  [680] = {x=33.236, y=0.000, z=-5.463, rx=-0.000, ry=0.000, rz=-0.000, shoulder=lefty, elbow=epositive, wrist=wnegative, fatherId=fReference[0]}
  [681] = {x=32.701, y=0.000, z=-5.454, rx=-0.000, ry=0.000, rz=-0.000, shoulder=lefty, elbow=epositive, wrist=wnegative, fatherId=fReference[0]}
  [682] = {x=32.182, y=0.000, z=-5.451, rx=-0.000, ry=0.000, rz=-0.000, shoulder=lefty, elbow=epositive, wrist=wnegative, fatherId=fReference[0]}
  [683] = {x=31.672, y=0.000, z=-5.452, rx=-0.000, ry=0.000, rz=-0.000, shoulder=lefty, elbow=epositive, wrist=wnegative, fatherId=fReference[0]}
  [684] = {x=31.165, y=0.000, z=-5.456, rx=-0.000, ry=0.000, rz=-0.000, shoulder=lefty, elbow=epositive, wrist=wnegative, fatherId=fReference[0]}
  [685] = {x=30.661, y=0.000, z=-5.462, rx=-0.000, ry=0.000, rz=-0.000, shoulder=lefty, elbow=epositive, wrist=wnegative, fatherId=fReference[0]}
  [686] = {x=30.158, y=0.000, z=-5.467, rx=-0.000, ry=0.000, rz=-0.000, shoulder=lefty, elbow=epositive, wrist=wnegative, fatherId=fReference[0]}
  [687] = {x=29.655, y=0.000, z=-5.473, rx=-0.000, ry=0.000, rz=-0.000, shoulder=lefty, elbow=epositive, wrist=wnegative, fatherId=fReference[0]}
  [688] = {x=29.154, y=0.000, z=-5.480, rx=-0.000, ry=0.000, rz=-0.000, shoulder=lefty, elbow=epositive, wrist=wnegative, fatherId=fReference[0]}
  [689] = {x=28.652, y=0.000, z=-5.487, rx=-0.000, ry=0.000, rz=-0.000, shoulder=lefty, elbow=epositive, wrist=wnegative, fatherId=fReference[0]}
  [690] = {x=28.151, y=0.000, z=-5.494, rx=-0.000, ry=0.000, rz=-0.000, shoulder=lefty, elbow=epositive, wrist=wnegative, fatherId=fReference[0]}
  [691] = {x=27.650, y=0.000, z=-5.502, rx=-0.000, ry=0.000, rz=-0.000, shoulder=lefty, elbow=epositive, wrist=wnegative, fatherId=fReference[0]}
  [692] = {x=27.149, y=0.000, z=-5.510, rx=-0.000, ry=0.000, rz=-0.000, shoulder=lefty, elbow=epositive, wrist=wnegative, fatherId=fReference[0]}
  [693] = {x=26.649, y=0.000, z=-5.518, rx=-0.000, ry=0.000, rz=-0.000, shoulder=lefty, elbow=epositive, wrist=wnegative, fatherId=fReference[0]}
  [694] = {x=26.149, y=0.000, z=-5.526, rx=-0.000, ry=0.000, rz=-0.000, shoulder=lefty, elbow=epositive, wrist=wnegative, fatherId=fReference[0]}
  [695] = {x=25.648, y=0.000, z=-5.534, rx=-0.000, ry=0.000, rz=-0.000, shoulder=lefty, elbow=epositive, wrist=wnegative, fatherId=fReference[0]}
  [696] = {x=25.148, y=0.000, z=-5.543, rx=-0.000, ry=0.000, rz=-0.000, shoulder=lefty, elbow=epositive, wrist=wnegative, fatherId=fReference[0]}
  [697] = {x=24.648, y=0.000, z=-5.551, rx=-0.000, ry=0.000, rz=-0.000, shoulder=lefty, elbow=epositive, wrist=wnegative, fatherId=fReference[0]}
  [698] = {x=24.148, y=0.000, z=-5.559, rx=-0.000, ry=0.000, rz=-0.000, shoulder=lefty, elbow=epositive, wrist=wnegative, fatherId=fReference[0]}
  [699] = {x=23.647, y=0.000, z=-5.568, rx=-0.000, ry=0.000, rz=-0.000, shoulder=lefty, elbow=epositive, wrist=wnegative, fatherId=fReference[0]}
  [700] = {x=23.147, y=0.000, z=-5.576, rx=-0.000, ry=0.000, rz=-0.000, shoulder=lefty, elbow=epositive, wrist=wnegative, fatherId=fReference[0]}
  [701] = {x=22.647, y=0.000, z=-5.585, rx=-0.000, ry=0.000, rz=-0.000, shoulder=lefty, elbow=epositive, wrist=wnegative, fatherId=fReference[0]}
  [702] = {x=22.147, y=0.000, z=-5.594, rx=-0.000, ry=0.000, rz=-0.000, shoulder=lefty, elbow=epositive, wrist=wnegative, fatherId=fReference[0]}
  [703] = {x=21.647, y=0.000, z=-5.602, rx=-0.000, ry=0.000, rz=-0.000, shoulder=lefty, elbow=epositive, wrist=wnegative, fatherId=fReference[0]}
  [704] = {x=21.146, y=0.000, z=-5.611, rx=-0.000, ry=0.000, rz=-0.000, shoulder=lefty, elbow=epositive, wrist=wnegative, fatherId=fReference[0]}
  [705] = {x=20.646, y=0.000, z=-5.620, rx=-0.000, ry=0.000, rz=-0.000, shoulder=lefty, elbow=epositive, wrist=wnegative, fatherId=fReference[0]}
  [706] = {x=20.146, y=0.000, z=-5.629, rx=-0.000, ry=0.000, rz=-0.000, shoulder=lefty, elbow=epositive, wrist=wnegative, fatherId=fReference[0]}
  [707] = {x=19.646, y=0.000, z=-5.638, rx=-0.000, ry=0.000, rz=-0.000, shoulder=lefty, elbow=epositive, wrist=wnegative, fatherId=fReference[0]}
  [708] = {x=19.146, y=0.000, z=-5.647, rx=-0.000, ry=0.000, rz=-0.000, shoulder=lefty, elbow=epositive, wrist=wnegative, fatherId=fReference[0]}
  [709] = {x=18.646, y=0.000, z=-5.656, rx=-0.000, ry=0.000, rz=-0.000, shoulder=lefty, elbow=epositive, wrist=wnegative, fatherId=fReference[0]}
  [710] = {x=18.145, y=0.000, z=-5.665, rx=-0.000, ry=0.000, rz=-0.000, shoulder=lefty, elbow=epositive, wrist=wnegative, fatherId=fReference[0]}
  [711] = {x=17.645, y=0.000, z=-5.675, rx=-0.000, ry=0.000, rz=-0.000, shoulder=lefty, elbow=epositive, wrist=wnegative, fatherId=fReference[0]}
  [712] = {x=17.145, y=0.000, z=-5.684, rx=-0.000, ry=0.000, rz=-0.000, shoulder=lefty, elbow=epositive, wrist=wnegative, fatherId=fReference[0]}
  [713] = {x=16.645, y=0.000, z=-5.693, rx=-0.000, ry=0.000, rz=-0.000, shoulder=lefty, elbow=epositive, wrist=wnegative, fatherId=fReference[0]}
  [714] = {x=16.144, y=0.000, z=-5.702, rx=-0.000, ry=0.000, rz=-0.000, shoulder=lefty, elbow=epositive, wrist=wnegative, fatherId=fReference[0]}
  [715] = {x=15.644, y=0.000, z=-5.712, rx=-0.000, ry=0.000, rz=-0.000, shoulder=lefty, elbow=epositive, wrist=wnegative, fatherId=fReference[0]}
  [716] = {x=15.144, y=0.000, z=-5.721, rx=-0.000, ry=0.000, rz=-0.000, shoulder=lefty, elbow=epositive, wrist=wnegative, fatherId=fReference[0]}
  [717] = {x=14.644, y=0.000, z=-5.730, rx=-0.000, ry=0.000, rz=-0.000, shoulder=lefty, elbow=epositive, wrist=wnegative, fatherId=fReference[0]}
  [718] = {x=14.144, y=0.000, z=-5.740, rx=-0.000, ry=0.000, rz=-0.000, shoulder=lefty, elbow=epositive, wrist=wnegative, fatherId=fReference[0]}
  [719] = {x=13.643, y=0.000, z=-5.749, rx=-0.000, ry=0.000, rz=-0.000, shoulder=lefty, elbow=epositive, wrist=wnegative, fatherId=fReference[0]}
  [720] = {x=13.143, y=0.000, z=-5.758, rx=-0.000, ry=0.000, rz=-0.000, shoulder=lefty, elbow=epositive, wrist=wnegative, fatherId=fReference[0]}
  [721] = {x=12.643, y=0.000, z=-5.767, rx=-0.000, ry=0.000, rz=-0.000, shoulder=lefty, elbow=epositive, wrist=wnegative, fatherId=fReference[0]}
  [722] = {x=12.142, y=0.000, z=-5.776, rx=-0.000, ry=0.000, rz=-0.000, shoulder=lefty, elbow=epositive, wrist=wnegative, fatherId=fReference[0]}
  [723] = {x=11.641, y=0.000, z=-5.785, rx=-0.000, ry=0.000, rz=-0.000, shoulder=lefty, elbow=epositive, wrist=wnegative, fatherId=fReference[0]}
  [724] = {x=11.141, y=0.000, z=-5.794, rx=-0.000, ry=0.000, rz=-0.000, shoulder=lefty, elbow=epositive, wrist=wnegative, fatherId=fReference[0]}
  [725] = {x=10.640, y=0.000, z=-5.803, rx=-0.000, ry=0.000, rz=-0.000, shoulder=lefty, elbow=epositive, wrist=wnegative, fatherId=fReference[0]}
  [726] = {x=10.139, y=0.000, z=-5.811, rx=-0.000, ry=0.000, rz=-0.000, shoulder=lefty, elbow=epositive, wrist=wnegative, fatherId=fReference[0]}
  [727] = {x=9.638, y=0.000, z=-5.820, rx=-0.000, ry=0.000, rz=-0.000, shoulder=lefty, elbow=epositive, wrist=wnegative, fatherId=fReference[0]}
  [728] = {x=9.137, y=0.000, z=-5.828, rx=-0.000, ry=0.000, rz=-0.000, shoulder=lefty, elbow=epositive, wrist=wnegative, fatherId=fReference[0]}
  [729] = {x=8.637, y=0.000, z=-5.837, rx=-0.000, ry=0.000, rz=-0.000, shoulder=lefty, elbow=epositive, wrist=wnegative, fatherId=fReference[0]}
  [730] = {x=8.136, y=0.000, z=-5.846, rx=-0.000, ry=0.000, rz=-0.000, shoulder=lefty, elbow=epositive, wrist=wnegative, fatherId=fReference[0]}
  [731] = {x=7.635, y=0.000, z=-5.854, rx=-0.000, ry=0.000, rz=-0.000, shoulder=lefty, elbow=epositive, wrist=wnegative, fatherId=fReference[0]}
  [732] = {x=7.134, y=0.000, z=-5.862, rx=-0.000, ry=0.000, rz=-0.000, shoulder=lefty, elbow=epositive, wrist=wnegative, fatherId=fReference[0]}
  [733] = {x=6.633, y=0.000, z=-5.870, rx=-0.000, ry=0.000, rz=-0.000, shoulder=lefty, elbow=epositive, wrist=wnegative, fatherId=fReference[0]}
  [734] = {x=6.131, y=0.000, z=-5.878, rx=-0.000, ry=0.000, rz=-0.000, shoulder=lefty, elbow=epositive, wrist=wnegative, fatherId=fReference[0]}
  [735] = {x=5.630, y=0.000, z=-5.886, rx=-0.000, ry=0.000, rz=-0.000, shoulder=lefty, elbow=epositive, wrist=wnegative, fatherId=fReference[0]}
  [736] = {x=5.128, y=0.000, z=-5.894, rx=-0.000, ry=0.000, rz=-0.000, shoulder=lefty, elbow=epositive, wrist=wnegative, fatherId=fReference[0]}
  [737] = {x=4.626, y=0.000, z=-5.902, rx=-0.000, ry=0.000, rz=-0.000, shoulder=lefty, elbow=epositive, wrist=wnegative, fatherId=fReference[0]}
  [738] = {x=4.123, y=0.000, z=-5.909, rx=-0.000, ry=0.000, rz=-0.000, shoulder=lefty, elbow=epositive, wrist=wnegative, fatherId=fReference[0]}
  [739] = {x=3.621, y=0.000, z=-5.917, rx=-0.000, ry=0.000, rz=-0.000, shoulder=lefty, elbow=epositive, wrist=wnegative, fatherId=fReference[0]}
  [740] = {x=3.120, y=0.000, z=-5.925, rx=-0.000, ry=0.000, rz=-0.000, shoulder=lefty, elbow=epositive, wrist=wnegative, fatherId=fReference[0]}
  [741] = {x=2.618, y=0.000, z=-5.932, rx=-0.000, ry=0.000, rz=-0.000, shoulder=lefty, elbow=epositive, wrist=wnegative, fatherId=fReference[0]}
  [742] = {x=2.117, y=0.000, z=-5.941, rx=-0.000, ry=0.000, rz=-0.000, shoulder=lefty, elbow=epositive, wrist=wnegative, fatherId=fReference[0]}
  [743] = {x=1.616, y=0.000, z=-5.949, rx=-0.000, ry=0.000, rz=-0.000, shoulder=lefty, elbow=epositive, wrist=wnegative, fatherId=fReference[0]}
  [744] = {x=1.114, y=0.000, z=-5.957, rx=-0.000, ry=0.000, rz=-0.000, shoulder=lefty, elbow=epositive, wrist=wnegative, fatherId=fReference[0]}
  [745] = {x=0.614, y=0.000, z=-5.966, rx=-0.000, ry=0.000, rz=-0.000, shoulder=lefty, elbow=epositive, wrist=wnegative, fatherId=fReference[0]}
  [746] = {x=0.112, y=0.000, z=-5.974, rx=-0.000, ry=0.000, rz=-0.000, shoulder=lefty, elbow=epositive, wrist=wnegative, fatherId=fReference[0]}
  [747] = {x=-0.389, y=0.000, z=-5.983, rx=-0.000, ry=0.000, rz=-0.000, shoulder=lefty, elbow=epositive, wrist=wnegative, fatherId=fReference[0]}
  [748] = {x=-0.890, y=0.000, z=-5.991, rx=-0.000, ry=0.000, rz=-0.000, shoulder=lefty, elbow=epositive, wrist=wnegative, fatherId=fReference[0]}
  [749] = {x=-1.392, y=0.000, z=-6.000, rx=-0.000, ry=0.000, rz=-0.000, shoulder=lefty, elbow=epositive, wrist=wnegative, fatherId=fReference[0]}
  [750] = {x=-1.893, y=0.000, z=-6.009, rx=-0.000, ry=0.000, rz=-0.000, shoulder=lefty, elbow=epositive, wrist=wnegative, fatherId=fReference[0]}
  [751] = {x=-2.394, y=0.000, z=-6.017, rx=-0.000, ry=0.000, rz=-0.000, shoulder=lefty, elbow=epositive, wrist=wnegative, fatherId=fReference[0]}
  [752] = {x=-2.895, y=0.000, z=-6.026, rx=-0.000, ry=0.000, rz=-0.000, shoulder=lefty, elbow=epositive, wrist=wnegative, fatherId=fReference[0]}
  [753] = {x=-3.397, y=0.000, z=-6.035, rx=-0.000, ry=0.000, rz=-0.000, shoulder=lefty, elbow=epositive, wrist=wnegative, fatherId=fReference[0]}
  [754] = {x=-3.898, y=0.000, z=-6.044, rx=-0.000, ry=0.000, rz=-0.000, shoulder=lefty, elbow=epositive, wrist=wnegative, fatherId=fReference[0]}
  [755] = {x=-4.399, y=0.000, z=-6.053, rx=-0.000, ry=0.000, rz=-0.000, shoulder=lefty, elbow=epositive, wrist=wnegative, fatherId=fReference[0]}
  [756] = {x=-4.901, y=0.000, z=-6.062, rx=-0.000, ry=0.000, rz=-0.000, shoulder=lefty, elbow=epositive, wrist=wnegative, fatherId=fReference[0]}
  [757] = {x=-5.402, y=0.000, z=-6.071, rx=-0.000, ry=0.000, rz=-0.000, shoulder=lefty, elbow=epositive, wrist=wnegative, fatherId=fReference[0]}
  [758] = {x=-5.902, y=0.000, z=-6.080, rx=-0.000, ry=0.000, rz=-0.000, shoulder=lefty, elbow=epositive, wrist=wnegative, fatherId=fReference[0]}
  [759] = {x=-6.404, y=0.000, z=-6.089, rx=-0.000, ry=0.000, rz=-0.000, shoulder=lefty, elbow=epositive, wrist=wnegative, fatherId=fReference[0]}
  [760] = {x=-6.906, y=0.000, z=-6.098, rx=-0.000, ry=0.000, rz=-0.000, shoulder=lefty, elbow=epositive, wrist=wnegative, fatherId=fReference[0]}
  [761] = {x=-7.407, y=0.000, z=-6.107, rx=-0.000, ry=0.000, rz=-0.000, shoulder=lefty, elbow=epositive, wrist=wnegative, fatherId=fReference[0]}
  [762] = {x=-7.907, y=0.000, z=-6.117, rx=-0.000, ry=0.000, rz=-0.000, shoulder=lefty, elbow=epositive, wrist=wnegative, fatherId=fReference[0]}
  [763] = {x=-8.409, y=0.000, z=-6.126, rx=-0.000, ry=0.000, rz=-0.000, shoulder=lefty, elbow=epositive, wrist=wnegative, fatherId=fReference[0]}
  [764] = {x=-8.910, y=0.000, z=-6.136, rx=-0.000, ry=0.000, rz=-0.000, shoulder=lefty, elbow=epositive, wrist=wnegative, fatherId=fReference[0]}
  [765] = {x=-9.411, y=0.000, z=-6.145, rx=-0.000, ry=0.000, rz=-0.000, shoulder=lefty, elbow=epositive, wrist=wnegative, fatherId=fReference[0]}
  [766] = {x=-9.912, y=0.000, z=-6.155, rx=-0.000, ry=0.000, rz=-0.000, shoulder=lefty, elbow=epositive, wrist=wnegative, fatherId=fReference[0]}
  [767] = {x=-10.412, y=0.000, z=-6.165, rx=-0.000, ry=0.000, rz=-0.000, shoulder=lefty, elbow=epositive, wrist=wnegative, fatherId=fReference[0]}
  [768] = {x=-10.913, y=0.000, z=-6.175, rx=-0.000, ry=0.000, rz=-0.000, shoulder=lefty, elbow=epositive, wrist=wnegative, fatherId=fReference[0]}
  [769] = {x=-11.413, y=0.000, z=-6.185, rx=-0.000, ry=0.000, rz=-0.000, shoulder=lefty, elbow=epositive, wrist=wnegative, fatherId=fReference[0]}
  [770] = {x=-11.914, y=0.000, z=-6.195, rx=-0.000, ry=0.000, rz=-0.000, shoulder=lefty, elbow=epositive, wrist=wnegative, fatherId=fReference[0]}
  [771] = {x=-12.414, y=0.000, z=-6.206, rx=-0.000, ry=0.000, rz=-0.000, shoulder=lefty, elbow=epositive, wrist=wnegative, fatherId=fReference[0]}
  [772] = {x=-12.916, y=0.000, z=-6.215, rx=-0.000, ry=0.000, rz=-0.000, shoulder=lefty, elbow=epositive, wrist=wnegative, fatherId=fReference[0]}
  [773] = {x=-13.416, y=0.000, z=-6.225, rx=-0.000, ry=0.000, rz=-0.000, shoulder=lefty, elbow=epositive, wrist=wnegative, fatherId=fReference[0]}
  [774] = {x=-13.916, y=0.000, z=-6.236, rx=-0.000, ry=0.000, rz=-0.000, shoulder=lefty, elbow=epositive, wrist=wnegative, fatherId=fReference[0]}
  [775] = {x=-14.417, y=0.000, z=-6.246, rx=-0.000, ry=0.000, rz=-0.000, shoulder=lefty, elbow=epositive, wrist=wnegative, fatherId=fReference[0]}
  [776] = {x=-14.916, y=0.000, z=-6.257, rx=-0.000, ry=0.000, rz=-0.000, shoulder=lefty, elbow=epositive, wrist=wnegative, fatherId=fReference[0]}
  [777] = {x=-15.418, y=0.000, z=-6.267, rx=-0.000, ry=0.000, rz=-0.000, shoulder=lefty, elbow=epositive, wrist=wnegative, fatherId=fReference[0]}
  [778] = {x=-15.917, y=0.000, z=-6.278, rx=-0.000, ry=0.000, rz=-0.000, shoulder=lefty, elbow=epositive, wrist=wnegative, fatherId=fReference[0]}
  [779] = {x=-16.418, y=0.000, z=-6.288, rx=-0.000, ry=0.000, rz=-0.000, shoulder=lefty, elbow=epositive, wrist=wnegative, fatherId=fReference[0]}
  [780] = {x=-16.918, y=0.000, z=-6.300, rx=-0.000, ry=0.000, rz=-0.000, shoulder=lefty, elbow=epositive, wrist=wnegative, fatherId=fReference[0]}
  [781] = {x=-17.419, y=0.000, z=-6.310, rx=-0.000, ry=0.000, rz=-0.000, shoulder=lefty, elbow=epositive, wrist=wnegative, fatherId=fReference[0]}
  [782] = {x=-17.919, y=0.000, z=-6.321, rx=-0.000, ry=0.000, rz=-0.000, shoulder=lefty, elbow=epositive, wrist=wnegative, fatherId=fReference[0]}
  [783] = {x=-18.420, y=0.000, z=-6.331, rx=-0.000, ry=0.000, rz=-0.000, shoulder=lefty, elbow=epositive, wrist=wnegative, fatherId=fReference[0]}
  [784] = {x=-18.920, y=0.000, z=-6.342, rx=-0.000, ry=0.000, rz=-0.000, shoulder=lefty, elbow=epositive, wrist=wnegative, fatherId=fReference[0]}
  [785] = {x=-19.418, y=0.000, z=-6.354, rx=-0.000, ry=0.000, rz=-0.000, shoulder=lefty, elbow=epositive, wrist=wnegative, fatherId=fReference[0]}
  [786] = {x=-19.920, y=0.000, z=-6.364, rx=-0.000, ry=0.000, rz=-0.000, shoulder=lefty, elbow=epositive, wrist=wnegative, fatherId=fReference[0]}
  [787] = {x=-20.420, y=0.000, z=-6.375, rx=-0.000, ry=0.000, rz=-0.000, shoulder=lefty, elbow=epositive, wrist=wnegative, fatherId=fReference[0]}
  [788] = {x=-20.920, y=0.000, z=-6.386, rx=-0.000, ry=0.000, rz=-0.000, shoulder=lefty, elbow=epositive, wrist=wnegative, fatherId=fReference[0]}
  [789] = {x=-21.421, y=0.000, z=-6.397, rx=-0.000, ry=0.000, rz=-0.000, shoulder=lefty, elbow=epositive, wrist=wnegative, fatherId=fReference[0]}
  [790] = {x=-21.922, y=0.000, z=-6.407, rx=-0.000, ry=0.000, rz=-0.000, shoulder=lefty, elbow=epositive, wrist=wnegative, fatherId=fReference[0]}
  [791] = {x=-22.422, y=0.000, z=-6.418, rx=-0.000, ry=0.000, rz=-0.000, shoulder=lefty, elbow=epositive, wrist=wnegative, fatherId=fReference[0]}
  [792] = {x=-22.921, y=0.000, z=-6.431, rx=-0.000, ry=0.000, rz=-0.000, shoulder=lefty, elbow=epositive, wrist=wnegative, fatherId=fReference[0]}
  [793] = {x=-23.422, y=0.000, z=-6.442, rx=-0.000, ry=0.000, rz=-0.000, shoulder=lefty, elbow=epositive, wrist=wnegative, fatherId=fReference[0]}
  [794] = {x=-23.924, y=0.000, z=-6.453, rx=-0.000, ry=0.000, rz=-0.000, shoulder=lefty, elbow=epositive, wrist=wnegative, fatherId=fReference[0]}
  [795] = {x=-24.426, y=0.000, z=-6.464, rx=-0.000, ry=0.000, rz=-0.000, shoulder=lefty, elbow=epositive, wrist=wnegative, fatherId=fReference[0]}
  [796] = {x=-24.927, y=0.000, z=-6.476, rx=-0.000, ry=0.000, rz=-0.000, shoulder=lefty, elbow=epositive, wrist=wnegative, fatherId=fReference[0]}
  [797] = {x=-25.427, y=0.000, z=-6.488, rx=-0.000, ry=0.000, rz=-0.000, shoulder=lefty, elbow=epositive, wrist=wnegative, fatherId=fReference[0]}
  [798] = {x=-25.928, y=0.000, z=-6.501, rx=-0.000, ry=0.000, rz=-0.000, shoulder=lefty, elbow=epositive, wrist=wnegative, fatherId=fReference[0]}
  [799] = {x=-26.428, y=0.000, z=-6.513, rx=-0.000, ry=0.000, rz=-0.000, shoulder=lefty, elbow=epositive, wrist=wnegative, fatherId=fReference[0]}
  [800] = {x=-26.930, y=0.000, z=-6.526, rx=-0.000, ry=0.000, rz=-0.000, shoulder=lefty, elbow=epositive, wrist=wnegative, fatherId=fReference[0]}
  [801] = {x=-27.433, y=0.000, z=-6.538, rx=-0.000, ry=0.000, rz=-0.000, shoulder=lefty, elbow=epositive, wrist=wnegative, fatherId=fReference[0]}
  [802] = {x=-27.936, y=0.000, z=-6.550, rx=-0.000, ry=0.000, rz=-0.000, shoulder=lefty, elbow=epositive, wrist=wnegative, fatherId=fReference[0]}
  [803] = {x=-28.441, y=0.000, z=-6.561, rx=-0.000, ry=0.000, rz=-0.000, shoulder=lefty, elbow=epositive, wrist=wnegative, fatherId=fReference[0]}
  [804] = {x=-28.947, y=0.000, z=-6.571, rx=-0.000, ry=0.000, rz=-0.000, shoulder=lefty, elbow=epositive, wrist=wnegative, fatherId=fReference[0]}
  [805] = {x=-29.456, y=0.000, z=-6.581, rx=-0.000, ry=0.000, rz=-0.000, shoulder=lefty, elbow=epositive, wrist=wnegative, fatherId=fReference[0]}
  [806] = {x=-29.968, y=0.000, z=-6.590, rx=-0.000, ry=0.000, rz=-0.000, shoulder=lefty, elbow=epositive, wrist=wnegative, fatherId=fReference[0]}
  [807] = {x=-30.478, y=0.000, z=-6.600, rx=-0.000, ry=0.000, rz=-0.000, shoulder=lefty, elbow=epositive, wrist=wnegative, fatherId=fReference[0]}
  [808] = {x=-30.992, y=0.000, z=-6.610, rx=-0.000, ry=0.000, rz=-0.000, shoulder=lefty, elbow=epositive, wrist=wnegative, fatherId=fReference[0]}
  [809] = {x=-31.504, y=0.000, z=-6.617, rx=-0.000, ry=0.000, rz=-0.000, shoulder=lefty, elbow=epositive, wrist=wnegative, fatherId=fReference[0]}
  [810] = {x=-31.724, y=0.000, z=-6.575, rx=-0.000, ry=0.000, rz=-0.000, shoulder=lefty, elbow=epositive, wrist=wnegative, fatherId=fReference[0]}
  [811] = {x=-31.202, y=0.000, z=-6.559, rx=-0.000, ry=0.000, rz=-0.000, shoulder=lefty, elbow=epositive, wrist=wnegative, fatherId=fReference[0]}
  [812] = {x=-30.687, y=0.000, z=-6.554, rx=-0.000, ry=0.000, rz=-0.000, shoulder=lefty, elbow=epositive, wrist=wnegative, fatherId=fReference[0]}
  [813] = {x=-30.181, y=0.000, z=-6.554, rx=-0.000, ry=0.000, rz=-0.000, shoulder=lefty, elbow=epositive, wrist=wnegative, fatherId=fReference[0]}
  [814] = {x=-29.680, y=0.000, z=-6.557, rx=-0.000, ry=0.000, rz=-0.000, shoulder=lefty, elbow=epositive, wrist=wnegative, fatherId=fReference[0]}
  [815] = {x=-29.180, y=0.000, z=-6.561, rx=-0.000, ry=0.000, rz=-0.000, shoulder=lefty, elbow=epositive, wrist=wnegative, fatherId=fReference[0]}
  [816] = {x=-28.680, y=0.000, z=-6.566, rx=-0.000, ry=0.000, rz=-0.000, shoulder=lefty, elbow=epositive, wrist=wnegative, fatherId=fReference[0]}
  [817] = {x=-28.180, y=0.000, z=-6.571, rx=-0.000, ry=0.000, rz=-0.000, shoulder=lefty, elbow=epositive, wrist=wnegative, fatherId=fReference[0]}
  [818] = {x=-27.680, y=0.000, z=-6.577, rx=-0.000, ry=0.000, rz=-0.000, shoulder=lefty, elbow=epositive, wrist=wnegative, fatherId=fReference[0]}
  [819] = {x=-27.180, y=0.000, z=-6.584, rx=-0.000, ry=0.000, rz=-0.000, shoulder=lefty, elbow=epositive, wrist=wnegative, fatherId=fReference[0]}
  [820] = {x=-26.679, y=0.000, z=-6.591, rx=-0.000, ry=0.000, rz=-0.000, shoulder=lefty, elbow=epositive, wrist=wnegative, fatherId=fReference[0]}
  [821] = {x=-26.178, y=0.000, z=-6.598, rx=-0.000, ry=0.000, rz=-0.000, shoulder=lefty, elbow=epositive, wrist=wnegative, fatherId=fReference[0]}
  [822] = {x=-25.677, y=0.000, z=-6.605, rx=-0.000, ry=0.000, rz=-0.000, shoulder=lefty, elbow=epositive, wrist=wnegative, fatherId=fReference[0]}
  [823] = {x=-25.175, y=0.000, z=-6.613, rx=-0.000, ry=0.000, rz=-0.000, shoulder=lefty, elbow=epositive, wrist=wnegative, fatherId=fReference[0]}
  [824] = {x=-24.675, y=0.000, z=-6.622, rx=-0.000, ry=0.000, rz=-0.000, shoulder=lefty, elbow=epositive, wrist=wnegative, fatherId=fReference[0]}
  [825] = {x=-24.174, y=0.000, z=-6.630, rx=-0.000, ry=0.000, rz=-0.000, shoulder=lefty, elbow=epositive, wrist=wnegative, fatherId=fReference[0]}
  [826] = {x=-23.672, y=0.000, z=-6.639, rx=-0.000, ry=0.000, rz=-0.000, shoulder=lefty, elbow=epositive, wrist=wnegative, fatherId=fReference[0]}
  [827] = {x=-23.171, y=0.000, z=-6.647, rx=-0.000, ry=0.000, rz=-0.000, shoulder=lefty, elbow=epositive, wrist=wnegative, fatherId=fReference[0]}
  [828] = {x=-22.670, y=0.000, z=-6.656, rx=-0.000, ry=0.000, rz=-0.000, shoulder=lefty, elbow=epositive, wrist=wnegative, fatherId=fReference[0]}
  [829] = {x=-22.168, y=0.000, z=-6.665, rx=-0.000, ry=0.000, rz=-0.000, shoulder=lefty, elbow=epositive, wrist=wnegative, fatherId=fReference[0]}
  [830] = {x=-21.666, y=0.000, z=-6.673, rx=-0.000, ry=0.000, rz=-0.000, shoulder=lefty, elbow=epositive, wrist=wnegative, fatherId=fReference[0]}
  [831] = {x=-21.165, y=0.000, z=-6.682, rx=-0.000, ry=0.000, rz=-0.000, shoulder=lefty, elbow=epositive, wrist=wnegative, fatherId=fReference[0]}
  [832] = {x=-20.664, y=0.000, z=-6.691, rx=-0.000, ry=0.000, rz=-0.000, shoulder=lefty, elbow=epositive, wrist=wnegative, fatherId=fReference[0]}
  [833] = {x=-20.162, y=0.000, z=-6.699, rx=-0.000, ry=0.000, rz=-0.000, shoulder=lefty, elbow=epositive, wrist=wnegative, fatherId=fReference[0]}
  [834] = {x=-19.661, y=0.000, z=-6.708, rx=-0.000, ry=0.000, rz=-0.000, shoulder=lefty, elbow=epositive, wrist=wnegative, fatherId=fReference[0]}
  [835] = {x=-19.159, y=0.000, z=-6.716, rx=-0.000, ry=0.000, rz=-0.000, shoulder=lefty, elbow=epositive, wrist=wnegative, fatherId=fReference[0]}
  [836] = {x=-18.657, y=0.000, z=-6.724, rx=-0.000, ry=0.000, rz=-0.000, shoulder=lefty, elbow=epositive, wrist=wnegative, fatherId=fReference[0]}
  [837] = {x=-18.156, y=0.000, z=-6.733, rx=-0.000, ry=0.000, rz=-0.000, shoulder=lefty, elbow=epositive, wrist=wnegative, fatherId=fReference[0]}
  [838] = {x=-17.654, y=0.000, z=-6.742, rx=-0.000, ry=0.000, rz=-0.000, shoulder=lefty, elbow=epositive, wrist=wnegative, fatherId=fReference[0]}
  [839] = {x=-17.152, y=0.000, z=-6.750, rx=-0.000, ry=0.000, rz=-0.000, shoulder=lefty, elbow=epositive, wrist=wnegative, fatherId=fReference[0]}
  [840] = {x=-16.651, y=0.000, z=-6.758, rx=-0.000, ry=0.000, rz=-0.000, shoulder=lefty, elbow=epositive, wrist=wnegative, fatherId=fReference[0]}
  [841] = {x=-16.149, y=0.000, z=-6.767, rx=-0.000, ry=0.000, rz=-0.000, shoulder=lefty, elbow=epositive, wrist=wnegative, fatherId=fReference[0]}
  [842] = {x=-15.647, y=0.000, z=-6.776, rx=-0.000, ry=0.000, rz=-0.000, shoulder=lefty, elbow=epositive, wrist=wnegative, fatherId=fReference[0]}
  [843] = {x=-15.146, y=0.000, z=-6.785, rx=-0.000, ry=0.000, rz=-0.000, shoulder=lefty, elbow=epositive, wrist=wnegative, fatherId=fReference[0]}
  [844] = {x=-14.643, y=0.000, z=-6.793, rx=-0.000, ry=0.000, rz=-0.000, shoulder=lefty, elbow=epositive, wrist=wnegative, fatherId=fReference[0]}
  [845] = {x=-14.141, y=0.000, z=-6.802, rx=-0.000, ry=0.000, rz=-0.000, shoulder=lefty, elbow=epositive, wrist=wnegative, fatherId=fReference[0]}
  [846] = {x=-13.639, y=0.000, z=-6.811, rx=-0.000, ry=0.000, rz=-0.000, shoulder=lefty, elbow=epositive, wrist=wnegative, fatherId=fReference[0]}
  [847] = {x=-13.138, y=0.000, z=-6.819, rx=-0.000, ry=0.000, rz=-0.000, shoulder=lefty, elbow=epositive, wrist=wnegative, fatherId=fReference[0]}
  [848] = {x=-12.636, y=0.000, z=-6.828, rx=-0.000, ry=0.000, rz=-0.000, shoulder=lefty, elbow=epositive, wrist=wnegative, fatherId=fReference[0]}
  [849] = {x=-12.134, y=0.000, z=-6.837, rx=-0.000, ry=0.000, rz=-0.000, shoulder=lefty, elbow=epositive, wrist=wnegative, fatherId=fReference[0]}
  [850] = {x=-11.632, y=0.000, z=-6.846, rx=-0.000, ry=0.000, rz=-0.000, shoulder=lefty, elbow=epositive, wrist=wnegative, fatherId=fReference[0]}
  [851] = {x=-11.130, y=0.000, z=-6.856, rx=-0.000, ry=0.000, rz=-0.000, shoulder=lefty, elbow=epositive, wrist=wnegative, fatherId=fReference[0]}
  [852] = {x=-10.627, y=0.000, z=-6.865, rx=-0.000, ry=0.000, rz=-0.000, shoulder=lefty, elbow=epositive, wrist=wnegative, fatherId=fReference[0]}
  [853] = {x=-10.124, y=0.000, z=-6.874, rx=-0.000, ry=0.000, rz=-0.000, shoulder=lefty, elbow=epositive, wrist=wnegative, fatherId=fReference[0]}
  [854] = {x=-9.622, y=0.000, z=-6.884, rx=-0.000, ry=0.000, rz=-0.000, shoulder=lefty, elbow=epositive, wrist=wnegative, fatherId=fReference[0]}
  [855] = {x=-9.120, y=0.000, z=-6.893, rx=-0.000, ry=0.000, rz=-0.000, shoulder=lefty, elbow=epositive, wrist=wnegative, fatherId=fReference[0]}
  [856] = {x=-8.617, y=0.000, z=-6.902, rx=-0.000, ry=0.000, rz=-0.000, shoulder=lefty, elbow=epositive, wrist=wnegative, fatherId=fReference[0]}
  [857] = {x=-8.114, y=0.000, z=-6.910, rx=-0.000, ry=0.000, rz=-0.000, shoulder=lefty, elbow=epositive, wrist=wnegative, fatherId=fReference[0]}
  [858] = {x=-7.611, y=0.000, z=-6.920, rx=-0.000, ry=0.000, rz=-0.000, shoulder=lefty, elbow=epositive, wrist=wnegative, fatherId=fReference[0]}
  [859] = {x=-7.109, y=0.000, z=-6.928, rx=-0.000, ry=0.000, rz=-0.000, shoulder=lefty, elbow=epositive, wrist=wnegative, fatherId=fReference[0]}
  [860] = {x=-6.606, y=0.000, z=-6.937, rx=-0.000, ry=0.000, rz=-0.000, shoulder=lefty, elbow=epositive, wrist=wnegative, fatherId=fReference[0]}
  [861] = {x=-6.104, y=0.000, z=-6.945, rx=-0.000, ry=0.000, rz=-0.000, shoulder=lefty, elbow=epositive, wrist=wnegative, fatherId=fReference[0]}
  [862] = {x=-5.601, y=0.000, z=-6.952, rx=-0.000, ry=0.000, rz=-0.000, shoulder=lefty, elbow=epositive, wrist=wnegative, fatherId=fReference[0]}
  [863] = {x=-5.099, y=0.000, z=-6.961, rx=-0.000, ry=0.000, rz=-0.000, shoulder=lefty, elbow=epositive, wrist=wnegative, fatherId=fReference[0]}
  [864] = {x=-4.597, y=0.000, z=-6.969, rx=-0.000, ry=0.000, rz=-0.000, shoulder=lefty, elbow=epositive, wrist=wnegative, fatherId=fReference[0]}
  [865] = {x=-4.094, y=0.000, z=-6.976, rx=-0.000, ry=0.000, rz=-0.000, shoulder=lefty, elbow=epositive, wrist=wnegative, fatherId=fReference[0]}
  [866] = {x=-3.592, y=0.000, z=-6.985, rx=-0.000, ry=0.000, rz=-0.000, shoulder=lefty, elbow=epositive, wrist=wnegative, fatherId=fReference[0]}
  [867] = {x=-3.090, y=0.000, z=-6.993, rx=-0.000, ry=0.000, rz=-0.000, shoulder=lefty, elbow=epositive, wrist=wnegative, fatherId=fReference[0]}
  [868] = {x=-2.587, y=0.000, z=-7.001, rx=-0.000, ry=0.000, rz=-0.000, shoulder=lefty, elbow=epositive, wrist=wnegative, fatherId=fReference[0]}
  [869] = {x=-2.084, y=0.000, z=-7.009, rx=-0.000, ry=0.000, rz=-0.000, shoulder=lefty, elbow=epositive, wrist=wnegative, fatherId=fReference[0]}
  [870] = {x=-1.581, y=0.000, z=-7.016, rx=-0.000, ry=0.000, rz=-0.000, shoulder=lefty, elbow=epositive, wrist=wnegative, fatherId=fReference[0]}
  [871] = {x=-1.078, y=0.000, z=-7.025, rx=-0.000, ry=0.000, rz=-0.000, shoulder=lefty, elbow=epositive, wrist=wnegative, fatherId=fReference[0]}
  [872] = {x=-0.576, y=0.000, z=-7.034, rx=-0.000, ry=0.000, rz=-0.000, shoulder=lefty, elbow=epositive, wrist=wnegative, fatherId=fReference[0]}
  [873] = {x=-0.073, y=0.000, z=-7.042, rx=-0.000, ry=0.000, rz=-0.000, shoulder=lefty, elbow=epositive, wrist=wnegative, fatherId=fReference[0]}
  [874] = {x=0.430, y=0.000, z=-7.050, rx=-0.000, ry=0.000, rz=-0.000, shoulder=lefty, elbow=epositive, wrist=wnegative, fatherId=fReference[0]}
  [875] = {x=0.933, y=0.000, z=-7.058, rx=-0.000, ry=0.000, rz=-0.000, shoulder=lefty, elbow=epositive, wrist=wnegative, fatherId=fReference[0]}
  [876] = {x=1.436, y=0.000, z=-7.067, rx=-0.000, ry=0.000, rz=-0.000, shoulder=lefty, elbow=epositive, wrist=wnegative, fatherId=fReference[0]}
  [877] = {x=1.939, y=0.000, z=-7.076, rx=-0.000, ry=0.000, rz=-0.000, shoulder=lefty, elbow=epositive, wrist=wnegative, fatherId=fReference[0]}
  [878] = {x=2.442, y=0.000, z=-7.085, rx=-0.000, ry=0.000, rz=-0.000, shoulder=lefty, elbow=epositive, wrist=wnegative, fatherId=fReference[0]}
  [879] = {x=2.945, y=0.000, z=-7.093, rx=-0.000, ry=0.000, rz=-0.000, shoulder=lefty, elbow=epositive, wrist=wnegative, fatherId=fReference[0]}
  [880] = {x=3.448, y=0.000, z=-7.102, rx=-0.000, ry=0.000, rz=-0.000, shoulder=lefty, elbow=epositive, wrist=wnegative, fatherId=fReference[0]}
  [881] = {x=3.951, y=0.000, z=-7.112, rx=-0.000, ry=0.000, rz=-0.000, shoulder=lefty, elbow=epositive, wrist=wnegative, fatherId=fReference[0]}
  [882] = {x=4.454, y=0.000, z=-7.121, rx=-0.000, ry=0.000, rz=-0.000, shoulder=lefty, elbow=epositive, wrist=wnegative, fatherId=fReference[0]}
  [883] = {x=4.957, y=0.000, z=-7.129, rx=-0.000, ry=0.000, rz=-0.000, shoulder=lefty, elbow=epositive, wrist=wnegative, fatherId=fReference[0]}
  [884] = {x=5.460, y=0.000, z=-7.138, rx=-0.000, ry=0.000, rz=-0.000, shoulder=lefty, elbow=epositive, wrist=wnegative, fatherId=fReference[0]}
  [885] = {x=5.963, y=0.000, z=-7.147, rx=-0.000, ry=0.000, rz=-0.000, shoulder=lefty, elbow=epositive, wrist=wnegative, fatherId=fReference[0]}
  [886] = {x=6.466, y=0.000, z=-7.157, rx=-0.000, ry=0.000, rz=-0.000, shoulder=lefty, elbow=epositive, wrist=wnegative, fatherId=fReference[0]}
  [887] = {x=6.968, y=0.000, z=-7.167, rx=-0.000, ry=0.000, rz=-0.000, shoulder=lefty, elbow=epositive, wrist=wnegative, fatherId=fReference[0]}
  [888] = {x=7.471, y=0.000, z=-7.176, rx=-0.000, ry=0.000, rz=-0.000, shoulder=lefty, elbow=epositive, wrist=wnegative, fatherId=fReference[0]}
  [889] = {x=7.975, y=0.000, z=-7.186, rx=-0.000, ry=0.000, rz=-0.000, shoulder=lefty, elbow=epositive, wrist=wnegative, fatherId=fReference[0]}
  [890] = {x=8.478, y=0.000, z=-7.196, rx=-0.000, ry=0.000, rz=-0.000, shoulder=lefty, elbow=epositive, wrist=wnegative, fatherId=fReference[0]}
  [891] = {x=8.981, y=0.000, z=-7.205, rx=-0.000, ry=0.000, rz=-0.000, shoulder=lefty, elbow=epositive, wrist=wnegative, fatherId=fReference[0]}
  [892] = {x=9.484, y=0.000, z=-7.215, rx=-0.000, ry=0.000, rz=-0.000, shoulder=lefty, elbow=epositive, wrist=wnegative, fatherId=fReference[0]}
  [893] = {x=9.986, y=0.000, z=-7.225, rx=-0.000, ry=0.000, rz=-0.000, shoulder=lefty, elbow=epositive, wrist=wnegative, fatherId=fReference[0]}
  [894] = {x=10.489, y=0.000, z=-7.236, rx=-0.000, ry=0.000, rz=-0.000, shoulder=lefty, elbow=epositive, wrist=wnegative, fatherId=fReference[0]}
  [895] = {x=10.991, y=0.000, z=-7.246, rx=-0.000, ry=0.000, rz=-0.000, shoulder=lefty, elbow=epositive, wrist=wnegative, fatherId=fReference[0]}
  [896] = {x=11.494, y=0.000, z=-7.256, rx=-0.000, ry=0.000, rz=-0.000, shoulder=lefty, elbow=epositive, wrist=wnegative, fatherId=fReference[0]}
  [897] = {x=11.998, y=0.000, z=-7.267, rx=-0.000, ry=0.000, rz=-0.000, shoulder=lefty, elbow=epositive, wrist=wnegative, fatherId=fReference[0]}
  [898] = {x=12.500, y=0.000, z=-7.277, rx=-0.000, ry=0.000, rz=-0.000, shoulder=lefty, elbow=epositive, wrist=wnegative, fatherId=fReference[0]}
  [899] = {x=13.003, y=0.000, z=-7.287, rx=-0.000, ry=0.000, rz=-0.000, shoulder=lefty, elbow=epositive, wrist=wnegative, fatherId=fReference[0]}
  [900] = {x=13.506, y=0.000, z=-7.298, rx=-0.000, ry=0.000, rz=-0.000, shoulder=lefty, elbow=epositive, wrist=wnegative, fatherId=fReference[0]}
  [901] = {x=14.010, y=0.000, z=-7.308, rx=-0.000, ry=0.000, rz=-0.000, shoulder=lefty, elbow=epositive, wrist=wnegative, fatherId=fReference[0]}
  [902] = {x=14.513, y=0.000, z=-7.319, rx=-0.000, ry=0.000, rz=-0.000, shoulder=lefty, elbow=epositive, wrist=wnegative, fatherId=fReference[0]}
  [903] = {x=15.017, y=0.000, z=-7.330, rx=-0.000, ry=0.000, rz=-0.000, shoulder=lefty, elbow=epositive, wrist=wnegative, fatherId=fReference[0]}
  [904] = {x=15.519, y=0.000, z=-7.341, rx=-0.000, ry=0.000, rz=-0.000, shoulder=lefty, elbow=epositive, wrist=wnegative, fatherId=fReference[0]}
  [905] = {x=16.024, y=0.000, z=-7.350, rx=-0.000, ry=0.000, rz=-0.000, shoulder=lefty, elbow=epositive, wrist=wnegative, fatherId=fReference[0]}
  [906] = {x=16.527, y=0.000, z=-7.361, rx=-0.000, ry=0.000, rz=-0.000, shoulder=lefty, elbow=epositive, wrist=wnegative, fatherId=fReference[0]}
  [907] = {x=17.030, y=0.000, z=-7.373, rx=-0.000, ry=0.000, rz=-0.000, shoulder=lefty, elbow=epositive, wrist=wnegative, fatherId=fReference[0]}
  [908] = {x=17.534, y=0.000, z=-7.383, rx=-0.000, ry=0.000, rz=-0.000, shoulder=lefty, elbow=epositive, wrist=wnegative, fatherId=fReference[0]}
  [909] = {x=18.037, y=0.000, z=-7.394, rx=-0.000, ry=0.000, rz=-0.000, shoulder=lefty, elbow=epositive, wrist=wnegative, fatherId=fReference[0]}
  [910] = {x=18.542, y=0.000, z=-7.405, rx=-0.000, ry=0.000, rz=-0.000, shoulder=lefty, elbow=epositive, wrist=wnegative, fatherId=fReference[0]}
  [911] = {x=19.046, y=0.000, z=-7.415, rx=-0.000, ry=0.000, rz=-0.000, shoulder=lefty, elbow=epositive, wrist=wnegative, fatherId=fReference[0]}
  [912] = {x=19.550, y=0.000, z=-7.428, rx=-0.000, ry=0.000, rz=-0.000, shoulder=lefty, elbow=epositive, wrist=wnegative, fatherId=fReference[0]}
  [913] = {x=20.055, y=0.000, z=-7.437, rx=-0.000, ry=0.000, rz=-0.000, shoulder=lefty, elbow=epositive, wrist=wnegative, fatherId=fReference[0]}
  [914] = {x=20.559, y=0.000, z=-7.450, rx=-0.000, ry=0.000, rz=-0.000, shoulder=lefty, elbow=epositive, wrist=wnegative, fatherId=fReference[0]}
  [915] = {x=21.062, y=0.000, z=-7.462, rx=-0.000, ry=0.000, rz=-0.000, shoulder=lefty, elbow=epositive, wrist=wnegative, fatherId=fReference[0]}
  [916] = {x=21.567, y=0.000, z=-7.473, rx=-0.000, ry=0.000, rz=-0.000, shoulder=lefty, elbow=epositive, wrist=wnegative, fatherId=fReference[0]}
  [917] = {x=22.072, y=0.000, z=-7.484, rx=-0.000, ry=0.000, rz=-0.000, shoulder=lefty, elbow=epositive, wrist=wnegative, fatherId=fReference[0]}
  [918] = {x=22.578, y=0.000, z=-7.493, rx=-0.000, ry=0.000, rz=-0.000, shoulder=lefty, elbow=epositive, wrist=wnegative, fatherId=fReference[0]}
  [919] = {x=23.082, y=0.000, z=-7.505, rx=-0.000, ry=0.000, rz=-0.000, shoulder=lefty, elbow=epositive, wrist=wnegative, fatherId=fReference[0]}
  [920] = {x=23.588, y=0.000, z=-7.515, rx=-0.000, ry=0.000, rz=-0.000, shoulder=lefty, elbow=epositive, wrist=wnegative, fatherId=fReference[0]}
  [921] = {x=24.093, y=0.000, z=-7.528, rx=-0.000, ry=0.000, rz=-0.000, shoulder=lefty, elbow=epositive, wrist=wnegative, fatherId=fReference[0]}
  [922] = {x=24.598, y=0.000, z=-7.540, rx=-0.000, ry=0.000, rz=-0.000, shoulder=lefty, elbow=epositive, wrist=wnegative, fatherId=fReference[0]}
  [923] = {x=25.104, y=0.000, z=-7.552, rx=-0.000, ry=0.000, rz=-0.000, shoulder=lefty, elbow=epositive, wrist=wnegative, fatherId=fReference[0]}
  [924] = {x=25.610, y=0.000, z=-7.563, rx=-0.000, ry=0.000, rz=-0.000, shoulder=lefty, elbow=epositive, wrist=wnegative, fatherId=fReference[0]}
  [925] = {x=26.118, y=0.000, z=-7.572, rx=-0.000, ry=0.000, rz=-0.000, shoulder=lefty, elbow=epositive, wrist=wnegative, fatherId=fReference[0]}
  [926] = {x=26.625, y=0.000, z=-7.583, rx=-0.000, ry=0.000, rz=-0.000, shoulder=lefty, elbow=epositive, wrist=wnegative, fatherId=fReference[0]}
  [927] = {x=27.133, y=0.000, z=-7.595, rx=-0.000, ry=0.000, rz=-0.000, shoulder=lefty, elbow=epositive, wrist=wnegative, fatherId=fReference[0]}
  [928] = {x=27.642, y=0.000, z=-7.608, rx=-0.000, ry=0.000, rz=-0.000, shoulder=lefty, elbow=epositive, wrist=wnegative, fatherId=fReference[0]}
  [929] = {x=28.150, y=0.000, z=-7.621, rx=-0.000, ry=0.000, rz=-0.000, shoulder=lefty, elbow=epositive, wrist=wnegative, fatherId=fReference[0]}
  [930] = {x=28.660, y=0.000, z=-7.635, rx=-0.000, ry=0.000, rz=-0.000, shoulder=lefty, elbow=epositive, wrist=wnegative, fatherId=fReference[0]}
  [931] = {x=29.171, y=0.000, z=-7.649, rx=-0.000, ry=0.000, rz=-0.000, shoulder=lefty, elbow=epositive, wrist=wnegative, fatherId=fReference[0]}
  [932] = {x=29.687, y=0.000, z=-7.662, rx=-0.000, ry=0.000, rz=-0.000, shoulder=lefty, elbow=epositive, wrist=wnegative, fatherId=fReference[0]}
  [933] = {x=30.201, y=0.000, z=-7.676, rx=-0.000, ry=0.000, rz=-0.000, shoulder=lefty, elbow=epositive, wrist=wnegative, fatherId=fReference[0]}
  [934] = {x=30.718, y=0.000, z=-7.689, rx=-0.000, ry=0.000, rz=-0.000, shoulder=lefty, elbow=epositive, wrist=wnegative, fatherId=fReference[0]}
  [935] = {x=31.236, y=0.000, z=-7.703, rx=-0.000, ry=0.000, rz=-0.000, shoulder=lefty, elbow=epositive, wrist=wnegative, fatherId=fReference[0]}
  [936] = {x=31.759, y=0.000, z=-7.711, rx=-0.000, ry=0.000, rz=-0.000, shoulder=lefty, elbow=epositive, wrist=wnegative, fatherId=fReference[0]}
  [937] = {x=32.284, y=0.000, z=-7.720, rx=-0.000, ry=0.000, rz=-0.000, shoulder=lefty, elbow=epositive, wrist=wnegative, fatherId=fReference[0]}
  [938] = {x=32.364, y=0.000, z=-7.683, rx=-0.000, ry=0.000, rz=-0.000, shoulder=lefty, elbow=epositive, wrist=wnegative, fatherId=fReference[0]}
  [939] = {x=31.798, y=0.000, z=-7.661, rx=-0.000, ry=0.000, rz=-0.000, shoulder=lefty, elbow=epositive, wrist=wnegative, fatherId=fReference[0]}
  [940] = {x=31.266, y=0.000, z=-7.649, rx=-0.000, ry=0.000, rz=-0.000, shoulder=lefty, elbow=epositive, wrist=wnegative, fatherId=fReference[0]}
  [941] = {x=30.750, y=0.000, z=-7.644, rx=-0.000, ry=0.000, rz=-0.000, shoulder=lefty, elbow=epositive, wrist=wnegative, fatherId=fReference[0]}
  [942] = {x=30.241, y=0.000, z=-7.644, rx=-0.000, ry=0.000, rz=-0.000, shoulder=lefty, elbow=epositive, wrist=wnegative, fatherId=fReference[0]}
  [943] = {x=29.733, y=0.000, z=-7.645, rx=-0.000, ry=0.000, rz=-0.000, shoulder=lefty, elbow=epositive, wrist=wnegative, fatherId=fReference[0]}
  [944] = {x=29.227, y=0.000, z=-7.648, rx=-0.000, ry=0.000, rz=-0.000, shoulder=lefty, elbow=epositive, wrist=wnegative, fatherId=fReference[0]}
  [945] = {x=28.722, y=0.000, z=-7.652, rx=-0.000, ry=0.000, rz=-0.000, shoulder=lefty, elbow=epositive, wrist=wnegative, fatherId=fReference[0]}
  [946] = {x=28.218, y=0.000, z=-7.657, rx=-0.000, ry=0.000, rz=-0.000, shoulder=lefty, elbow=epositive, wrist=wnegative, fatherId=fReference[0]}
  [947] = {x=27.713, y=0.000, z=-7.663, rx=-0.000, ry=0.000, rz=-0.000, shoulder=lefty, elbow=epositive, wrist=wnegative, fatherId=fReference[0]}
  [948] = {x=27.210, y=0.000, z=-7.670, rx=-0.000, ry=0.000, rz=-0.000, shoulder=lefty, elbow=epositive, wrist=wnegative, fatherId=fReference[0]}
  [949] = {x=26.709, y=0.000, z=-7.677, rx=-0.000, ry=0.000, rz=-0.000, shoulder=lefty, elbow=epositive, wrist=wnegative, fatherId=fReference[0]}
  [950] = {x=26.207, y=0.000, z=-7.684, rx=-0.000, ry=0.000, rz=-0.000, shoulder=lefty, elbow=epositive, wrist=wnegative, fatherId=fReference[0]}
  [951] = {x=25.706, y=0.000, z=-7.691, rx=-0.000, ry=0.000, rz=-0.000, shoulder=lefty, elbow=epositive, wrist=wnegative, fatherId=fReference[0]}
  [952] = {x=25.204, y=0.000, z=-7.699, rx=-0.000, ry=0.000, rz=-0.000, shoulder=lefty, elbow=epositive, wrist=wnegative, fatherId=fReference[0]}
  [953] = {x=24.703, y=0.000, z=-7.707, rx=-0.000, ry=0.000, rz=-0.000, shoulder=lefty, elbow=epositive, wrist=wnegative, fatherId=fReference[0]}
  [954] = {x=24.201, y=0.000, z=-7.715, rx=-0.000, ry=0.000, rz=-0.000, shoulder=lefty, elbow=epositive, wrist=wnegative, fatherId=fReference[0]}
  [955] = {x=23.699, y=0.000, z=-7.725, rx=-0.000, ry=0.000, rz=-0.000, shoulder=lefty, elbow=epositive, wrist=wnegative, fatherId=fReference[0]}
  [956] = {x=23.198, y=0.000, z=-7.734, rx=-0.000, ry=0.000, rz=-0.000, shoulder=lefty, elbow=epositive, wrist=wnegative, fatherId=fReference[0]}
  [957] = {x=22.699, y=0.000, z=-7.744, rx=-0.000, ry=0.000, rz=-0.000, shoulder=lefty, elbow=epositive, wrist=wnegative, fatherId=fReference[0]}
  [958] = {x=22.200, y=0.000, z=-7.752, rx=-0.000, ry=0.000, rz=-0.000, shoulder=lefty, elbow=epositive, wrist=wnegative, fatherId=fReference[0]}
  [959] = {x=21.699, y=0.000, z=-7.761, rx=-0.000, ry=0.000, rz=-0.000, shoulder=lefty, elbow=epositive, wrist=wnegative, fatherId=fReference[0]}
  [960] = {x=21.198, y=0.000, z=-7.770, rx=-0.000, ry=0.000, rz=-0.000, shoulder=lefty, elbow=epositive, wrist=wnegative, fatherId=fReference[0]}
  [961] = {x=20.698, y=0.000, z=-7.779, rx=-0.000, ry=0.000, rz=-0.000, shoulder=lefty, elbow=epositive, wrist=wnegative, fatherId=fReference[0]}
  [962] = {x=20.196, y=0.000, z=-7.789, rx=-0.000, ry=0.000, rz=-0.000, shoulder=lefty, elbow=epositive, wrist=wnegative, fatherId=fReference[0]}
  [963] = {x=19.696, y=0.000, z=-7.798, rx=-0.000, ry=0.000, rz=-0.000, shoulder=lefty, elbow=epositive, wrist=wnegative, fatherId=fReference[0]}
  [964] = {x=19.196, y=0.000, z=-7.808, rx=-0.000, ry=0.000, rz=-0.000, shoulder=lefty, elbow=epositive, wrist=wnegative, fatherId=fReference[0]}
  [965] = {x=18.696, y=0.000, z=-7.818, rx=-0.000, ry=0.000, rz=-0.000, shoulder=lefty, elbow=epositive, wrist=wnegative, fatherId=fReference[0]}
  [966] = {x=18.197, y=0.000, z=-7.828, rx=-0.000, ry=0.000, rz=-0.000, shoulder=lefty, elbow=epositive, wrist=wnegative, fatherId=fReference[0]}
  [967] = {x=17.695, y=0.000, z=-7.837, rx=-0.000, ry=0.000, rz=-0.000, shoulder=lefty, elbow=epositive, wrist=wnegative, fatherId=fReference[0]}
  [968] = {x=17.195, y=0.000, z=-7.847, rx=-0.000, ry=0.000, rz=-0.000, shoulder=lefty, elbow=epositive, wrist=wnegative, fatherId=fReference[0]}
  [969] = {x=16.696, y=0.000, z=-7.857, rx=-0.000, ry=0.000, rz=-0.000, shoulder=lefty, elbow=epositive, wrist=wnegative, fatherId=fReference[0]}
  [970] = {x=16.195, y=0.000, z=-7.867, rx=-0.000, ry=0.000, rz=-0.000, shoulder=lefty, elbow=epositive, wrist=wnegative, fatherId=fReference[0]}
  [971] = {x=15.694, y=0.000, z=-7.876, rx=-0.000, ry=0.000, rz=-0.000, shoulder=lefty, elbow=epositive, wrist=wnegative, fatherId=fReference[0]}
  [972] = {x=15.193, y=0.000, z=-7.886, rx=-0.000, ry=0.000, rz=-0.000, shoulder=lefty, elbow=epositive, wrist=wnegative, fatherId=fReference[0]}
  [973] = {x=14.693, y=0.000, z=-7.896, rx=-0.000, ry=0.000, rz=-0.000, shoulder=lefty, elbow=epositive, wrist=wnegative, fatherId=fReference[0]}
  [974] = {x=14.193, y=0.000, z=-7.906, rx=-0.000, ry=0.000, rz=-0.000, shoulder=lefty, elbow=epositive, wrist=wnegative, fatherId=fReference[0]}
  [975] = {x=13.693, y=0.000, z=-7.917, rx=-0.000, ry=0.000, rz=-0.000, shoulder=lefty, elbow=epositive, wrist=wnegative, fatherId=fReference[0]}
  [976] = {x=13.193, y=0.000, z=-7.926, rx=-0.000, ry=0.000, rz=-0.000, shoulder=lefty, elbow=epositive, wrist=wnegative, fatherId=fReference[0]}
  [977] = {x=12.693, y=0.000, z=-7.936, rx=-0.000, ry=0.000, rz=-0.000, shoulder=lefty, elbow=epositive, wrist=wnegative, fatherId=fReference[0]}
  [978] = {x=12.192, y=0.000, z=-7.945, rx=-0.000, ry=0.000, rz=-0.000, shoulder=lefty, elbow=epositive, wrist=wnegative, fatherId=fReference[0]}
  [979] = {x=11.692, y=0.000, z=-7.955, rx=-0.000, ry=0.000, rz=-0.000, shoulder=lefty, elbow=epositive, wrist=wnegative, fatherId=fReference[0]}
  [980] = {x=11.191, y=0.000, z=-7.964, rx=-0.000, ry=0.000, rz=-0.000, shoulder=lefty, elbow=epositive, wrist=wnegative, fatherId=fReference[0]}
  [981] = {x=10.689, y=0.000, z=-7.974, rx=-0.000, ry=0.000, rz=-0.000, shoulder=lefty, elbow=epositive, wrist=wnegative, fatherId=fReference[0]}
  [982] = {x=10.188, y=0.000, z=-7.983, rx=-0.000, ry=0.000, rz=-0.000, shoulder=lefty, elbow=epositive, wrist=wnegative, fatherId=fReference[0]}
  [983] = {x=9.686, y=0.000, z=-7.992, rx=-0.000, ry=0.000, rz=-0.000, shoulder=lefty, elbow=epositive, wrist=wnegative, fatherId=fReference[0]}
  [984] = {x=9.184, y=0.000, z=-8.001, rx=-0.000, ry=0.000, rz=-0.000, shoulder=lefty, elbow=epositive, wrist=wnegative, fatherId=fReference[0]}
  [985] = {x=8.683, y=0.000, z=-8.010, rx=-0.000, ry=0.000, rz=-0.000, shoulder=lefty, elbow=epositive, wrist=wnegative, fatherId=fReference[0]}
  [986] = {x=8.182, y=0.000, z=-8.020, rx=-0.000, ry=0.000, rz=-0.000, shoulder=lefty, elbow=epositive, wrist=wnegative, fatherId=fReference[0]}
  [987] = {x=7.679, y=0.000, z=-8.028, rx=-0.000, ry=0.000, rz=-0.000, shoulder=lefty, elbow=epositive, wrist=wnegative, fatherId=fReference[0]}
  [988] = {x=7.176, y=0.000, z=-8.036, rx=-0.000, ry=0.000, rz=-0.000, shoulder=lefty, elbow=epositive, wrist=wnegative, fatherId=fReference[0]}
  [989] = {x=6.673, y=0.000, z=-8.044, rx=-0.000, ry=0.000, rz=-0.000, shoulder=lefty, elbow=epositive, wrist=wnegative, fatherId=fReference[0]}
  [990] = {x=6.168, y=0.000, z=-8.050, rx=-0.000, ry=0.000, rz=-0.000, shoulder=lefty, elbow=epositive, wrist=wnegative, fatherId=fReference[0]}
  [991] = {x=5.665, y=0.000, z=-8.057, rx=-0.000, ry=0.000, rz=-0.000, shoulder=lefty, elbow=epositive, wrist=wnegative, fatherId=fReference[0]}
  [992] = {x=5.161, y=0.000, z=-8.065, rx=-0.000, ry=0.000, rz=-0.000, shoulder=lefty, elbow=epositive, wrist=wnegative, fatherId=fReference[0]}
  [993] = {x=4.658, y=0.000, z=-8.073, rx=-0.000, ry=0.000, rz=-0.000, shoulder=lefty, elbow=epositive, wrist=wnegative, fatherId=fReference[0]}
  [994] = {x=4.155, y=0.000, z=-8.081, rx=-0.000, ry=0.000, rz=-0.000, shoulder=lefty, elbow=epositive, wrist=wnegative, fatherId=fReference[0]}
  [995] = {x=3.651, y=0.000, z=-8.089, rx=-0.000, ry=0.000, rz=-0.000, shoulder=lefty, elbow=epositive, wrist=wnegative, fatherId=fReference[0]}
  [996] = {x=3.148, y=0.000, z=-8.097, rx=-0.000, ry=0.000, rz=-0.000, shoulder=lefty, elbow=epositive, wrist=wnegative, fatherId=fReference[0]}
  [997] = {x=2.644, y=0.000, z=-8.106, rx=-0.000, ry=0.000, rz=-0.000, shoulder=lefty, elbow=epositive, wrist=wnegative, fatherId=fReference[0]}
  [998] = {x=2.140, y=0.000, z=-8.114, rx=-0.000, ry=0.000, rz=-0.000, shoulder=lefty, elbow=epositive, wrist=wnegative, fatherId=fReference[0]}
  [999] = {x=1.637, y=0.000, z=-8.123, rx=-0.000, ry=0.000, rz=-0.000, shoulder=lefty, elbow=epositive, wrist=wnegative, fatherId=fReference[0]}
  [1000] = {x=1.135, y=0.000, z=-8.132, rx=-0.000, ry=0.000, rz=-0.000, shoulder=lefty, elbow=epositive, wrist=wnegative, fatherId=fReference[0]}
  [1001] = {x=0.632, y=0.000, z=-8.141, rx=-0.000, ry=0.000, rz=-0.000, shoulder=lefty, elbow=epositive, wrist=wnegative, fatherId=fReference[0]}
  [1002] = {x=0.128, y=0.000, z=-8.150, rx=-0.000, ry=0.000, rz=-0.000, shoulder=lefty, elbow=epositive, wrist=wnegative, fatherId=fReference[0]}
  [1003] = {x=-0.375, y=0.000, z=-8.160, rx=-0.000, ry=0.000, rz=-0.000, shoulder=lefty, elbow=epositive, wrist=wnegative, fatherId=fReference[0]}
  [1004] = {x=-0.877, y=0.000, z=-8.169, rx=-0.000, ry=0.000, rz=-0.000, shoulder=lefty, elbow=epositive, wrist=wnegative, fatherId=fReference[0]}
  [1005] = {x=-1.379, y=0.000, z=-8.178, rx=-0.000, ry=0.000, rz=-0.000, shoulder=lefty, elbow=epositive, wrist=wnegative, fatherId=fReference[0]}
  [1006] = {x=-1.881, y=0.000, z=-8.188, rx=-0.000, ry=0.000, rz=-0.000, shoulder=lefty, elbow=epositive, wrist=wnegative, fatherId=fReference[0]}
  [1007] = {x=-2.383, y=0.000, z=-8.198, rx=-0.000, ry=0.000, rz=-0.000, shoulder=lefty, elbow=epositive, wrist=wnegative, fatherId=fReference[0]}
  [1008] = {x=-2.885, y=0.000, z=-8.208, rx=-0.000, ry=0.000, rz=-0.000, shoulder=lefty, elbow=epositive, wrist=wnegative, fatherId=fReference[0]}
  [1009] = {x=-3.386, y=0.000, z=-8.218, rx=-0.000, ry=0.000, rz=-0.000, shoulder=lefty, elbow=epositive, wrist=wnegative, fatherId=fReference[0]}
  [1010] = {x=-3.888, y=0.000, z=-8.228, rx=-0.000, ry=0.000, rz=-0.000, shoulder=lefty, elbow=epositive, wrist=wnegative, fatherId=fReference[0]}
  [1011] = {x=-4.387, y=0.000, z=-8.238, rx=-0.000, ry=0.000, rz=-0.000, shoulder=lefty, elbow=epositive, wrist=wnegative, fatherId=fReference[0]}
  [1012] = {x=-4.890, y=0.000, z=-8.248, rx=-0.000, ry=0.000, rz=-0.000, shoulder=lefty, elbow=epositive, wrist=wnegative, fatherId=fReference[0]}
  [1013] = {x=-5.389, y=0.000, z=-8.258, rx=-0.000, ry=0.000, rz=-0.000, shoulder=lefty, elbow=epositive, wrist=wnegative, fatherId=fReference[0]}
  [1014] = {x=-5.892, y=0.000, z=-8.268, rx=-0.000, ry=0.000, rz=-0.000, shoulder=lefty, elbow=epositive, wrist=wnegative, fatherId=fReference[0]}
  [1015] = {x=-6.394, y=0.000, z=-8.278, rx=-0.000, ry=0.000, rz=-0.000, shoulder=lefty, elbow=epositive, wrist=wnegative, fatherId=fReference[0]}
  [1016] = {x=-6.892, y=0.000, z=-8.289, rx=-0.000, ry=0.000, rz=-0.000, shoulder=lefty, elbow=epositive, wrist=wnegative, fatherId=fReference[0]}
  [1017] = {x=-7.394, y=0.000, z=-8.299, rx=-0.000, ry=0.000, rz=-0.000, shoulder=lefty, elbow=epositive, wrist=wnegative, fatherId=fReference[0]}
  [1018] = {x=-7.894, y=0.000, z=-8.309, rx=-0.000, ry=0.000, rz=-0.000, shoulder=lefty, elbow=epositive, wrist=wnegative, fatherId=fReference[0]}
  [1019] = {x=-8.397, y=0.000, z=-8.319, rx=-0.000, ry=0.000, rz=-0.000, shoulder=lefty, elbow=epositive, wrist=wnegative, fatherId=fReference[0]}
  [1020] = {x=-8.896, y=0.000, z=-8.329, rx=-0.000, ry=0.000, rz=-0.000, shoulder=lefty, elbow=epositive, wrist=wnegative, fatherId=fReference[0]}
  [1021] = {x=-9.398, y=0.000, z=-8.339, rx=-0.000, ry=0.000, rz=-0.000, shoulder=lefty, elbow=epositive, wrist=wnegative, fatherId=fReference[0]}
  [1022] = {x=-9.898, y=0.000, z=-8.350, rx=-0.000, ry=0.000, rz=-0.000, shoulder=lefty, elbow=epositive, wrist=wnegative, fatherId=fReference[0]}
  [1023] = {x=-10.401, y=0.000, z=-8.360, rx=-0.000, ry=0.000, rz=-0.000, shoulder=lefty, elbow=epositive, wrist=wnegative, fatherId=fReference[0]}
  [1024] = {x=-10.901, y=0.000, z=-8.371, rx=-0.000, ry=0.000, rz=-0.000, shoulder=lefty, elbow=epositive, wrist=wnegative, fatherId=fReference[0]}
  [1025] = {x=-11.403, y=0.000, z=-8.380, rx=-0.000, ry=0.000, rz=-0.000, shoulder=lefty, elbow=epositive, wrist=wnegative, fatherId=fReference[0]}
  [1026] = {x=-11.906, y=0.000, z=-8.390, rx=-0.000, ry=0.000, rz=-0.000, shoulder=lefty, elbow=epositive, wrist=wnegative, fatherId=fReference[0]}
  [1027] = {x=-12.406, y=0.000, z=-8.401, rx=-0.000, ry=0.000, rz=-0.000, shoulder=lefty, elbow=epositive, wrist=wnegative, fatherId=fReference[0]}
  [1028] = {x=-12.909, y=0.000, z=-8.411, rx=-0.000, ry=0.000, rz=-0.000, shoulder=lefty, elbow=epositive, wrist=wnegative, fatherId=fReference[0]}
  [1029] = {x=-13.409, y=0.000, z=-8.421, rx=-0.000, ry=0.000, rz=-0.000, shoulder=lefty, elbow=epositive, wrist=wnegative, fatherId=fReference[0]}
  [1030] = {x=-13.913, y=0.000, z=-8.431, rx=-0.000, ry=0.000, rz=-0.000, shoulder=lefty, elbow=epositive, wrist=wnegative, fatherId=fReference[0]}
  [1031] = {x=-14.414, y=0.000, z=-8.441, rx=-0.000, ry=0.000, rz=-0.000, shoulder=lefty, elbow=epositive, wrist=wnegative, fatherId=fReference[0]}
  [1032] = {x=-14.918, y=0.000, z=-8.450, rx=-0.000, ry=0.000, rz=-0.000, shoulder=lefty, elbow=epositive, wrist=wnegative, fatherId=fReference[0]}
  [1033] = {x=-15.421, y=0.000, z=-8.460, rx=-0.000, ry=0.000, rz=-0.000, shoulder=lefty, elbow=epositive, wrist=wnegative, fatherId=fReference[0]}
  [1034] = {x=-15.924, y=0.000, z=-8.470, rx=-0.000, ry=0.000, rz=-0.000, shoulder=lefty, elbow=epositive, wrist=wnegative, fatherId=fReference[0]}
  [1035] = {x=-16.426, y=0.000, z=-8.481, rx=-0.000, ry=0.000, rz=-0.000, shoulder=lefty, elbow=epositive, wrist=wnegative, fatherId=fReference[0]}
  [1036] = {x=-16.929, y=0.000, z=-8.492, rx=-0.000, ry=0.000, rz=-0.000, shoulder=lefty, elbow=epositive, wrist=wnegative, fatherId=fReference[0]}
  [1037] = {x=-17.432, y=0.000, z=-8.502, rx=-0.000, ry=0.000, rz=-0.000, shoulder=lefty, elbow=epositive, wrist=wnegative, fatherId=fReference[0]}
  [1038] = {x=-17.935, y=0.000, z=-8.513, rx=-0.000, ry=0.000, rz=-0.000, shoulder=lefty, elbow=epositive, wrist=wnegative, fatherId=fReference[0]}
  [1039] = {x=-18.435, y=0.000, z=-8.525, rx=-0.000, ry=0.000, rz=-0.000, shoulder=lefty, elbow=epositive, wrist=wnegative, fatherId=fReference[0]}
  [1040] = {x=-18.938, y=0.000, z=-8.537, rx=-0.000, ry=0.000, rz=-0.000, shoulder=lefty, elbow=epositive, wrist=wnegative, fatherId=fReference[0]}
  [1041] = {x=-19.441, y=0.000, z=-8.549, rx=-0.000, ry=0.000, rz=-0.000, shoulder=lefty, elbow=epositive, wrist=wnegative, fatherId=fReference[0]}
  [1042] = {x=-19.943, y=0.000, z=-8.560, rx=-0.000, ry=0.000, rz=-0.000, shoulder=lefty, elbow=epositive, wrist=wnegative, fatherId=fReference[0]}
  [1043] = {x=-20.447, y=0.000, z=-8.571, rx=-0.000, ry=0.000, rz=-0.000, shoulder=lefty, elbow=epositive, wrist=wnegative, fatherId=fReference[0]}
  [1044] = {x=-20.948, y=0.000, z=-8.584, rx=-0.000, ry=0.000, rz=-0.000, shoulder=lefty, elbow=epositive, wrist=wnegative, fatherId=fReference[0]}
  [1045] = {x=-21.453, y=0.000, z=-8.595, rx=-0.000, ry=0.000, rz=-0.000, shoulder=lefty, elbow=epositive, wrist=wnegative, fatherId=fReference[0]}
  [1046] = {x=-21.954, y=0.000, z=-8.607, rx=-0.000, ry=0.000, rz=-0.000, shoulder=lefty, elbow=epositive, wrist=wnegative, fatherId=fReference[0]}
  [1047] = {x=-22.456, y=0.000, z=-8.620, rx=-0.000, ry=0.000, rz=-0.000, shoulder=lefty, elbow=epositive, wrist=wnegative, fatherId=fReference[0]}
  [1048] = {x=-22.960, y=0.000, z=-8.633, rx=-0.000, ry=0.000, rz=-0.000, shoulder=lefty, elbow=epositive, wrist=wnegative, fatherId=fReference[0]}
  [1049] = {x=-23.464, y=0.000, z=-8.646, rx=-0.000, ry=0.000, rz=-0.000, shoulder=lefty, elbow=epositive, wrist=wnegative, fatherId=fReference[0]}
  [1050] = {x=-23.968, y=0.000, z=-8.658, rx=-0.000, ry=0.000, rz=-0.000, shoulder=lefty, elbow=epositive, wrist=wnegative, fatherId=fReference[0]}
  [1051] = {x=-24.472, y=0.000, z=-8.671, rx=-0.000, ry=0.000, rz=-0.000, shoulder=lefty, elbow=epositive, wrist=wnegative, fatherId=fReference[0]}
  [1052] = {x=-24.975, y=0.000, z=-8.684, rx=-0.000, ry=0.000, rz=-0.000, shoulder=lefty, elbow=epositive, wrist=wnegative, fatherId=fReference[0]}
  [1053] = {x=-25.480, y=0.000, z=-8.697, rx=-0.000, ry=0.000, rz=-0.000, shoulder=lefty, elbow=epositive, wrist=wnegative, fatherId=fReference[0]}
  [1054] = {x=-25.984, y=0.000, z=-8.711, rx=-0.000, ry=0.000, rz=-0.000, shoulder=lefty, elbow=epositive, wrist=wnegative, fatherId=fReference[0]}
  [1055] = {x=-26.488, y=0.000, z=-8.726, rx=-0.000, ry=0.000, rz=-0.000, shoulder=lefty, elbow=epositive, wrist=wnegative, fatherId=fReference[0]}
  [1056] = {x=-26.991, y=0.000, z=-8.745, rx=-0.000, ry=0.000, rz=-0.000, shoulder=lefty, elbow=epositive, wrist=wnegative, fatherId=fReference[0]}
  [1057] = {x=-27.495, y=0.000, z=-8.763, rx=-0.000, ry=0.000, rz=-0.000, shoulder=lefty, elbow=epositive, wrist=wnegative, fatherId=fReference[0]}
  [1058] = {x=-27.999, y=0.000, z=-8.782, rx=-0.000, ry=0.000, rz=-0.000, shoulder=lefty, elbow=epositive, wrist=wnegative, fatherId=fReference[0]}
  [1059] = {x=-28.506, y=0.000, z=-8.801, rx=-0.000, ry=0.000, rz=-0.000, shoulder=lefty, elbow=epositive, wrist=wnegative, fatherId=fReference[0]}
  [1060] = {x=-29.016, y=0.000, z=-8.822, rx=-0.000, ry=0.000, rz=-0.000, shoulder=lefty, elbow=epositive, wrist=wnegative, fatherId=fReference[0]}
  [1061] = {x=-29.538, y=0.000, z=-8.842, rx=-0.000, ry=0.000, rz=-0.000, shoulder=lefty, elbow=epositive, wrist=wnegative, fatherId=fReference[0]}
  [1062] = {x=-30.064, y=0.000, z=-8.860, rx=-0.000, ry=0.000, rz=-0.000, shoulder=lefty, elbow=epositive, wrist=wnegative, fatherId=fReference[0]}
  [1063] = {x=-30.593, y=0.000, z=-8.872, rx=-0.000, ry=0.000, rz=-0.000, shoulder=lefty, elbow=epositive, wrist=wnegative, fatherId=fReference[0]}
  [1064] = {x=-30.649, y=0.000, z=-8.791, rx=-0.000, ry=0.000, rz=-0.000, shoulder=lefty, elbow=epositive, wrist=wnegative, fatherId=fReference[0]}
  [1065] = {x=-30.109, y=0.000, z=-8.751, rx=-0.000, ry=0.000, rz=-0.000, shoulder=lefty, elbow=epositive, wrist=wnegative, fatherId=fReference[0]}
  [1066] = {x=-29.603, y=0.000, z=-8.732, rx=-0.000, ry=0.000, rz=-0.000, shoulder=lefty, elbow=epositive, wrist=wnegative, fatherId=fReference[0]}
  [1067] = {x=-29.103, y=0.000, z=-8.717, rx=-0.000, ry=0.000, rz=-0.000, shoulder=lefty, elbow=epositive, wrist=wnegative, fatherId=fReference[0]}
  [1068] = {x=-28.604, y=0.000, z=-8.708, rx=-0.000, ry=0.000, rz=-0.000, shoulder=lefty, elbow=epositive, wrist=wnegative, fatherId=fReference[0]}
  [1069] = {x=-28.104, y=0.000, z=-8.703, rx=-0.000, ry=0.000, rz=-0.000, shoulder=lefty, elbow=epositive, wrist=wnegative, fatherId=fReference[0]}
  [1070] = {x=-27.602, y=0.000, z=-8.702, rx=-0.000, ry=0.000, rz=-0.000, shoulder=lefty, elbow=epositive, wrist=wnegative, fatherId=fReference[0]}
  [1071] = {x=-27.099, y=0.000, z=-8.704, rx=-0.000, ry=0.000, rz=-0.000, shoulder=lefty, elbow=epositive, wrist=wnegative, fatherId=fReference[0]}
  [1072] = {x=-26.596, y=0.000, z=-8.707, rx=-0.000, ry=0.000, rz=-0.000, shoulder=lefty, elbow=epositive, wrist=wnegative, fatherId=fReference[0]}
  [1073] = {x=-26.094, y=0.000, z=-8.712, rx=-0.000, ry=0.000, rz=-0.000, shoulder=lefty, elbow=epositive, wrist=wnegative, fatherId=fReference[0]}
  [1074] = {x=-25.592, y=0.000, z=-8.719, rx=-0.000, ry=0.000, rz=-0.000, shoulder=lefty, elbow=epositive, wrist=wnegative, fatherId=fReference[0]}
  [1075] = {x=-25.090, y=0.000, z=-8.726, rx=-0.000, ry=0.000, rz=-0.000, shoulder=lefty, elbow=epositive, wrist=wnegative, fatherId=fReference[0]}
  [1076] = {x=-24.588, y=0.000, z=-8.734, rx=-0.000, ry=0.000, rz=-0.000, shoulder=lefty, elbow=epositive, wrist=wnegative, fatherId=fReference[0]}
  [1077] = {x=-24.086, y=0.000, z=-8.742, rx=-0.000, ry=0.000, rz=-0.000, shoulder=lefty, elbow=epositive, wrist=wnegative, fatherId=fReference[0]}
  [1078] = {x=-23.583, y=0.000, z=-8.751, rx=-0.000, ry=0.000, rz=-0.000, shoulder=lefty, elbow=epositive, wrist=wnegative, fatherId=fReference[0]}
  [1079] = {x=-23.080, y=0.000, z=-8.760, rx=-0.000, ry=0.000, rz=-0.000, shoulder=lefty, elbow=epositive, wrist=wnegative, fatherId=fReference[0]}
  [1080] = {x=-22.578, y=0.000, z=-8.769, rx=-0.000, ry=0.000, rz=-0.000, shoulder=lefty, elbow=epositive, wrist=wnegative, fatherId=fReference[0]}
  [1081] = {x=-22.075, y=0.000, z=-8.778, rx=-0.000, ry=0.000, rz=-0.000, shoulder=lefty, elbow=epositive, wrist=wnegative, fatherId=fReference[0]}
  [1082] = {x=-21.571, y=0.000, z=-8.788, rx=-0.000, ry=0.000, rz=-0.000, shoulder=lefty, elbow=epositive, wrist=wnegative, fatherId=fReference[0]}
  [1083] = {x=-21.068, y=0.000, z=-8.798, rx=-0.000, ry=0.000, rz=-0.000, shoulder=lefty, elbow=epositive, wrist=wnegative, fatherId=fReference[0]}
  [1084] = {x=-20.566, y=0.000, z=-8.808, rx=-0.000, ry=0.000, rz=-0.000, shoulder=lefty, elbow=epositive, wrist=wnegative, fatherId=fReference[0]}
  [1085] = {x=-20.063, y=0.000, z=-8.818, rx=-0.000, ry=0.000, rz=-0.000, shoulder=lefty, elbow=epositive, wrist=wnegative, fatherId=fReference[0]}
  [1086] = {x=-19.560, y=0.000, z=-8.828, rx=-0.000, ry=0.000, rz=-0.000, shoulder=lefty, elbow=epositive, wrist=wnegative, fatherId=fReference[0]}
  [1087] = {x=-19.057, y=0.000, z=-8.839, rx=-0.000, ry=0.000, rz=-0.000, shoulder=lefty, elbow=epositive, wrist=wnegative, fatherId=fReference[0]}
  [1088] = {x=-18.554, y=0.000, z=-8.849, rx=-0.000, ry=0.000, rz=-0.000, shoulder=lefty, elbow=epositive, wrist=wnegative, fatherId=fReference[0]}
  [1089] = {x=-18.051, y=0.000, z=-8.860, rx=-0.000, ry=0.000, rz=-0.000, shoulder=lefty, elbow=epositive, wrist=wnegative, fatherId=fReference[0]}
  [1090] = {x=-17.548, y=0.000, z=-8.870, rx=-0.000, ry=0.000, rz=-0.000, shoulder=lefty, elbow=epositive, wrist=wnegative, fatherId=fReference[0]}
  [1091] = {x=-17.044, y=0.000, z=-8.880, rx=-0.000, ry=0.000, rz=-0.000, shoulder=lefty, elbow=epositive, wrist=wnegative, fatherId=fReference[0]}
  [1092] = {x=-16.541, y=0.000, z=-8.891, rx=-0.000, ry=0.000, rz=-0.000, shoulder=lefty, elbow=epositive, wrist=wnegative, fatherId=fReference[0]}
  [1093] = {x=-16.038, y=0.000, z=-8.901, rx=-0.000, ry=0.000, rz=-0.000, shoulder=lefty, elbow=epositive, wrist=wnegative, fatherId=fReference[0]}
  [1094] = {x=-15.535, y=0.000, z=-8.910, rx=-0.000, ry=0.000, rz=-0.000, shoulder=lefty, elbow=epositive, wrist=wnegative, fatherId=fReference[0]}
  [1095] = {x=-15.033, y=0.000, z=-8.920, rx=-0.000, ry=0.000, rz=-0.000, shoulder=lefty, elbow=epositive, wrist=wnegative, fatherId=fReference[0]}
  [1096] = {x=-14.531, y=0.000, z=-8.929, rx=-0.000, ry=0.000, rz=-0.000, shoulder=lefty, elbow=epositive, wrist=wnegative, fatherId=fReference[0]}
  [1097] = {x=-14.030, y=0.000, z=-8.938, rx=-0.000, ry=0.000, rz=-0.000, shoulder=lefty, elbow=epositive, wrist=wnegative, fatherId=fReference[0]}
  [1098] = {x=-13.527, y=0.000, z=-8.946, rx=-0.000, ry=0.000, rz=-0.000, shoulder=lefty, elbow=epositive, wrist=wnegative, fatherId=fReference[0]}
  [1099] = {x=-13.025, y=0.000, z=-8.955, rx=-0.000, ry=0.000, rz=-0.000, shoulder=lefty, elbow=epositive, wrist=wnegative, fatherId=fReference[0]}
  [1100] = {x=-12.523, y=0.000, z=-8.963, rx=-0.000, ry=0.000, rz=-0.000, shoulder=lefty, elbow=epositive, wrist=wnegative, fatherId=fReference[0]}
  [1101] = {x=-12.021, y=0.000, z=-8.972, rx=-0.000, ry=0.000, rz=-0.000, shoulder=lefty, elbow=epositive, wrist=wnegative, fatherId=fReference[0]}
  [1102] = {x=-11.518, y=0.000, z=-8.981, rx=-0.000, ry=0.000, rz=-0.000, shoulder=lefty, elbow=epositive, wrist=wnegative, fatherId=fReference[0]}
  [1103] = {x=-11.017, y=0.000, z=-8.990, rx=-0.000, ry=0.000, rz=-0.000, shoulder=lefty, elbow=epositive, wrist=wnegative, fatherId=fReference[0]}
  [1104] = {x=-10.514, y=0.000, z=-8.999, rx=-0.000, ry=0.000, rz=-0.000, shoulder=lefty, elbow=epositive, wrist=wnegative, fatherId=fReference[0]}
  [1105] = {x=-10.012, y=0.000, z=-9.007, rx=-0.000, ry=0.000, rz=-0.000, shoulder=lefty, elbow=epositive, wrist=wnegative, fatherId=fReference[0]}
  [1106] = {x=-9.510, y=0.000, z=-9.016, rx=-0.000, ry=0.000, rz=-0.000, shoulder=lefty, elbow=epositive, wrist=wnegative, fatherId=fReference[0]}
  [1107] = {x=-9.007, y=0.000, z=-9.025, rx=-0.000, ry=0.000, rz=-0.000, shoulder=lefty, elbow=epositive, wrist=wnegative, fatherId=fReference[0]}
  [1108] = {x=-8.505, y=0.000, z=-9.034, rx=-0.000, ry=0.000, rz=-0.000, shoulder=lefty, elbow=epositive, wrist=wnegative, fatherId=fReference[0]}
  [1109] = {x=-8.002, y=0.000, z=-9.042, rx=-0.000, ry=0.000, rz=-0.000, shoulder=lefty, elbow=epositive, wrist=wnegative, fatherId=fReference[0]}
  [1110] = {x=-7.500, y=0.000, z=-9.050, rx=-0.000, ry=0.000, rz=-0.000, shoulder=lefty, elbow=epositive, wrist=wnegative, fatherId=fReference[0]}
  [1111] = {x=-6.997, y=0.000, z=-9.059, rx=-0.000, ry=0.000, rz=-0.000, shoulder=lefty, elbow=epositive, wrist=wnegative, fatherId=fReference[0]}
  [1112] = {x=-6.495, y=0.000, z=-9.068, rx=-0.000, ry=0.000, rz=-0.000, shoulder=lefty, elbow=epositive, wrist=wnegative, fatherId=fReference[0]}
  [1113] = {x=-5.992, y=0.000, z=-9.076, rx=-0.000, ry=0.000, rz=-0.000, shoulder=lefty, elbow=epositive, wrist=wnegative, fatherId=fReference[0]}
  [1114] = {x=-5.490, y=0.000, z=-9.085, rx=-0.000, ry=0.000, rz=-0.000, shoulder=lefty, elbow=epositive, wrist=wnegative, fatherId=fReference[0]}
  [1115] = {x=-4.986, y=0.000, z=-9.093, rx=-0.000, ry=0.000, rz=-0.000, shoulder=lefty, elbow=epositive, wrist=wnegative, fatherId=fReference[0]}
  [1116] = {x=-4.483, y=0.000, z=-9.103, rx=-0.000, ry=0.000, rz=-0.000, shoulder=lefty, elbow=epositive, wrist=wnegative, fatherId=fReference[0]}
  [1117] = {x=-3.978, y=0.000, z=-9.111, rx=-0.000, ry=0.000, rz=-0.000, shoulder=lefty, elbow=epositive, wrist=wnegative, fatherId=fReference[0]}
  [1118] = {x=-3.475, y=0.000, z=-9.121, rx=-0.000, ry=0.000, rz=-0.000, shoulder=lefty, elbow=epositive, wrist=wnegative, fatherId=fReference[0]}
  [1119] = {x=-2.970, y=0.000, z=-9.129, rx=-0.000, ry=0.000, rz=-0.000, shoulder=lefty, elbow=epositive, wrist=wnegative, fatherId=fReference[0]}
  [1120] = {x=-2.465, y=0.000, z=-9.138, rx=-0.000, ry=0.000, rz=-0.000, shoulder=lefty, elbow=epositive, wrist=wnegative, fatherId=fReference[0]}
  [1121] = {x=-1.960, y=0.000, z=-9.147, rx=-0.000, ry=0.000, rz=-0.000, shoulder=lefty, elbow=epositive, wrist=wnegative, fatherId=fReference[0]}
  [1122] = {x=-1.455, y=0.000, z=-9.156, rx=-0.000, ry=0.000, rz=-0.000, shoulder=lefty, elbow=epositive, wrist=wnegative, fatherId=fReference[0]}
  [1123] = {x=-0.950, y=0.000, z=-9.165, rx=-0.000, ry=0.000, rz=-0.000, shoulder=lefty, elbow=epositive, wrist=wnegative, fatherId=fReference[0]}
  [1124] = {x=-0.445, y=0.000, z=-9.174, rx=-0.000, ry=0.000, rz=-0.000, shoulder=lefty, elbow=epositive, wrist=wnegative, fatherId=fReference[0]}
  [1125] = {x=0.061, y=0.000, z=-9.183, rx=-0.000, ry=0.000, rz=-0.000, shoulder=lefty, elbow=epositive, wrist=wnegative, fatherId=fReference[0]}
  [1126] = {x=0.566, y=0.000, z=-9.193, rx=-0.000, ry=0.000, rz=-0.000, shoulder=lefty, elbow=epositive, wrist=wnegative, fatherId=fReference[0]}
  [1127] = {x=1.071, y=0.000, z=-9.202, rx=-0.000, ry=0.000, rz=-0.000, shoulder=lefty, elbow=epositive, wrist=wnegative, fatherId=fReference[0]}
  [1128] = {x=1.576, y=0.000, z=-9.211, rx=-0.000, ry=0.000, rz=-0.000, shoulder=lefty, elbow=epositive, wrist=wnegative, fatherId=fReference[0]}
  [1129] = {x=2.079, y=0.000, z=-9.221, rx=-0.000, ry=0.000, rz=-0.000, shoulder=lefty, elbow=epositive, wrist=wnegative, fatherId=fReference[0]}
  [1130] = {x=2.584, y=0.000, z=-9.231, rx=-0.000, ry=0.000, rz=-0.000, shoulder=lefty, elbow=epositive, wrist=wnegative, fatherId=fReference[0]}
  [1131] = {x=3.088, y=0.000, z=-9.241, rx=-0.000, ry=0.000, rz=-0.000, shoulder=lefty, elbow=epositive, wrist=wnegative, fatherId=fReference[0]}
  [1132] = {x=3.592, y=0.000, z=-9.250, rx=-0.000, ry=0.000, rz=-0.000, shoulder=lefty, elbow=epositive, wrist=wnegative, fatherId=fReference[0]}
  [1133] = {x=4.096, y=0.000, z=-9.260, rx=-0.000, ry=0.000, rz=-0.000, shoulder=lefty, elbow=epositive, wrist=wnegative, fatherId=fReference[0]}
  [1134] = {x=4.600, y=0.000, z=-9.269, rx=-0.000, ry=0.000, rz=-0.000, shoulder=lefty, elbow=epositive, wrist=wnegative, fatherId=fReference[0]}
  [1135] = {x=5.104, y=0.000, z=-9.279, rx=-0.000, ry=0.000, rz=-0.000, shoulder=lefty, elbow=epositive, wrist=wnegative, fatherId=fReference[0]}
  [1136] = {x=5.608, y=0.000, z=-9.289, rx=-0.000, ry=0.000, rz=-0.000, shoulder=lefty, elbow=epositive, wrist=wnegative, fatherId=fReference[0]}
  [1137] = {x=6.111, y=0.000, z=-9.298, rx=-0.000, ry=0.000, rz=-0.000, shoulder=lefty, elbow=epositive, wrist=wnegative, fatherId=fReference[0]}
  [1138] = {x=6.612, y=0.000, z=-9.309, rx=-0.000, ry=0.000, rz=-0.000, shoulder=lefty, elbow=epositive, wrist=wnegative, fatherId=fReference[0]}
  [1139] = {x=7.118, y=0.000, z=-9.318, rx=-0.000, ry=0.000, rz=-0.000, shoulder=lefty, elbow=epositive, wrist=wnegative, fatherId=fReference[0]}
  [1140] = {x=7.621, y=0.000, z=-9.329, rx=-0.000, ry=0.000, rz=-0.000, shoulder=lefty, elbow=epositive, wrist=wnegative, fatherId=fReference[0]}
  [1141] = {x=8.125, y=0.000, z=-9.338, rx=-0.000, ry=0.000, rz=-0.000, shoulder=lefty, elbow=epositive, wrist=wnegative, fatherId=fReference[0]}
  [1142] = {x=8.629, y=0.000, z=-9.347, rx=-0.000, ry=0.000, rz=-0.000, shoulder=lefty, elbow=epositive, wrist=wnegative, fatherId=fReference[0]}
  [1143] = {x=9.132, y=0.000, z=-9.357, rx=-0.000, ry=0.000, rz=-0.000, shoulder=lefty, elbow=epositive, wrist=wnegative, fatherId=fReference[0]}
  [1144] = {x=9.635, y=0.000, z=-9.368, rx=-0.000, ry=0.000, rz=-0.000, shoulder=lefty, elbow=epositive, wrist=wnegative, fatherId=fReference[0]}
  [1145] = {x=10.139, y=0.000, z=-9.378, rx=-0.000, ry=0.000, rz=-0.000, shoulder=lefty, elbow=epositive, wrist=wnegative, fatherId=fReference[0]}
  [1146] = {x=10.642, y=0.000, z=-9.388, rx=-0.000, ry=0.000, rz=-0.000, shoulder=lefty, elbow=epositive, wrist=wnegative, fatherId=fReference[0]}
  [1147] = {x=11.145, y=0.000, z=-9.398, rx=-0.000, ry=0.000, rz=-0.000, shoulder=lefty, elbow=epositive, wrist=wnegative, fatherId=fReference[0]}
  [1148] = {x=11.649, y=0.000, z=-9.408, rx=-0.000, ry=0.000, rz=-0.000, shoulder=lefty, elbow=epositive, wrist=wnegative, fatherId=fReference[0]}
  [1149] = {x=12.152, y=0.000, z=-9.418, rx=-0.000, ry=0.000, rz=-0.000, shoulder=lefty, elbow=epositive, wrist=wnegative, fatherId=fReference[0]}
  [1150] = {x=12.656, y=0.000, z=-9.429, rx=-0.000, ry=0.000, rz=-0.000, shoulder=lefty, elbow=epositive, wrist=wnegative, fatherId=fReference[0]}
  [1151] = {x=13.161, y=0.000, z=-9.439, rx=-0.000, ry=0.000, rz=-0.000, shoulder=lefty, elbow=epositive, wrist=wnegative, fatherId=fReference[0]}
  [1152] = {x=13.665, y=0.000, z=-9.450, rx=-0.000, ry=0.000, rz=-0.000, shoulder=lefty, elbow=epositive, wrist=wnegative, fatherId=fReference[0]}
  [1153] = {x=14.170, y=0.000, z=-9.460, rx=-0.000, ry=0.000, rz=-0.000, shoulder=lefty, elbow=epositive, wrist=wnegative, fatherId=fReference[0]}
  [1154] = {x=14.673, y=0.000, z=-9.470, rx=-0.000, ry=0.000, rz=-0.000, shoulder=lefty, elbow=epositive, wrist=wnegative, fatherId=fReference[0]}
  [1155] = {x=15.178, y=0.000, z=-9.481, rx=-0.000, ry=0.000, rz=-0.000, shoulder=lefty, elbow=epositive, wrist=wnegative, fatherId=fReference[0]}
  [1156] = {x=15.683, y=0.000, z=-9.491, rx=-0.000, ry=0.000, rz=-0.000, shoulder=lefty, elbow=epositive, wrist=wnegative, fatherId=fReference[0]}
  [1157] = {x=16.188, y=0.000, z=-9.502, rx=-0.000, ry=0.000, rz=-0.000, shoulder=lefty, elbow=epositive, wrist=wnegative, fatherId=fReference[0]}
  [1158] = {x=16.693, y=0.000, z=-9.513, rx=-0.000, ry=0.000, rz=-0.000, shoulder=lefty, elbow=epositive, wrist=wnegative, fatherId=fReference[0]}
  [1159] = {x=17.198, y=0.000, z=-9.524, rx=-0.000, ry=0.000, rz=-0.000, shoulder=lefty, elbow=epositive, wrist=wnegative, fatherId=fReference[0]}
  [1160] = {x=17.705, y=0.000, z=-9.533, rx=-0.000, ry=0.000, rz=-0.000, shoulder=lefty, elbow=epositive, wrist=wnegative, fatherId=fReference[0]}
  [1161] = {x=18.212, y=0.000, z=-9.544, rx=-0.000, ry=0.000, rz=-0.000, shoulder=lefty, elbow=epositive, wrist=wnegative, fatherId=fReference[0]}
  [1162] = {x=18.718, y=0.000, z=-9.555, rx=-0.000, ry=0.000, rz=-0.000, shoulder=lefty, elbow=epositive, wrist=wnegative, fatherId=fReference[0]}
  [1163] = {x=19.225, y=0.000, z=-9.566, rx=-0.000, ry=0.000, rz=-0.000, shoulder=lefty, elbow=epositive, wrist=wnegative, fatherId=fReference[0]}
  [1164] = {x=19.732, y=0.000, z=-9.578, rx=-0.000, ry=0.000, rz=-0.000, shoulder=lefty, elbow=epositive, wrist=wnegative, fatherId=fReference[0]}
  [1165] = {x=20.239, y=0.000, z=-9.589, rx=-0.000, ry=0.000, rz=-0.000, shoulder=lefty, elbow=epositive, wrist=wnegative, fatherId=fReference[0]}
  [1166] = {x=20.746, y=0.000, z=-9.600, rx=-0.000, ry=0.000, rz=-0.000, shoulder=lefty, elbow=epositive, wrist=wnegative, fatherId=fReference[0]}
  [1167] = {x=21.253, y=0.000, z=-9.612, rx=-0.000, ry=0.000, rz=-0.000, shoulder=lefty, elbow=epositive, wrist=wnegative, fatherId=fReference[0]}
  [1168] = {x=21.761, y=0.000, z=-9.626, rx=-0.000, ry=0.000, rz=-0.000, shoulder=lefty, elbow=epositive, wrist=wnegative, fatherId=fReference[0]}
  [1169] = {x=22.271, y=0.000, z=-9.637, rx=-0.000, ry=0.000, rz=-0.000, shoulder=lefty, elbow=epositive, wrist=wnegative, fatherId=fReference[0]}
  [1170] = {x=22.778, y=0.000, z=-9.649, rx=-0.000, ry=0.000, rz=-0.000, shoulder=lefty, elbow=epositive, wrist=wnegative, fatherId=fReference[0]}
  [1171] = {x=23.289, y=0.000, z=-9.661, rx=-0.000, ry=0.000, rz=-0.000, shoulder=lefty, elbow=epositive, wrist=wnegative, fatherId=fReference[0]}
  [1172] = {x=23.797, y=0.000, z=-9.675, rx=-0.000, ry=0.000, rz=-0.000, shoulder=lefty, elbow=epositive, wrist=wnegative, fatherId=fReference[0]}
  [1173] = {x=24.306, y=0.000, z=-9.690, rx=-0.000, ry=0.000, rz=-0.000, shoulder=lefty, elbow=epositive, wrist=wnegative, fatherId=fReference[0]}
  [1174] = {x=24.816, y=0.000, z=-9.706, rx=-0.000, ry=0.000, rz=-0.000, shoulder=lefty, elbow=epositive, wrist=wnegative, fatherId=fReference[0]}
  [1175] = {x=25.326, y=0.000, z=-9.722, rx=-0.000, ry=0.000, rz=-0.000, shoulder=lefty, elbow=epositive, wrist=wnegative, fatherId=fReference[0]}
  [1176] = {x=25.838, y=0.000, z=-9.740, rx=-0.000, ry=0.000, rz=-0.000, shoulder=lefty, elbow=epositive, wrist=wnegative, fatherId=fReference[0]}
  [1177] = {x=26.351, y=0.000, z=-9.756, rx=-0.000, ry=0.000, rz=-0.000, shoulder=lefty, elbow=epositive, wrist=wnegative, fatherId=fReference[0]}
  [1178] = {x=26.863, y=0.000, z=-9.775, rx=-0.000, ry=0.000, rz=-0.000, shoulder=lefty, elbow=epositive, wrist=wnegative, fatherId=fReference[0]}
  [1179] = {x=27.379, y=0.000, z=-9.795, rx=-0.000, ry=0.000, rz=-0.000, shoulder=lefty, elbow=epositive, wrist=wnegative, fatherId=fReference[0]}
  [1180] = {x=27.895, y=0.000, z=-9.814, rx=-0.000, ry=0.000, rz=-0.000, shoulder=lefty, elbow=epositive, wrist=wnegative, fatherId=fReference[0]}
  [1181] = {x=28.414, y=0.000, z=-9.834, rx=-0.000, ry=0.000, rz=-0.000, shoulder=lefty, elbow=epositive, wrist=wnegative, fatherId=fReference[0]}
  [1182] = {x=28.938, y=0.000, z=-9.857, rx=-0.000, ry=0.000, rz=-0.000, shoulder=lefty, elbow=epositive, wrist=wnegative, fatherId=fReference[0]}
  [1183] = {x=29.467, y=0.000, z=-9.880, rx=-0.000, ry=0.000, rz=-0.000, shoulder=lefty, elbow=epositive, wrist=wnegative, fatherId=fReference[0]}
  [1184] = {x=30.006, y=0.000, z=-9.905, rx=-0.000, ry=0.000, rz=-0.000, shoulder=lefty, elbow=epositive, wrist=wnegative, fatherId=fReference[0]}
  [1185] = {x=30.553, y=0.000, z=-9.930, rx=-0.000, ry=0.000, rz=-0.000, shoulder=lefty, elbow=epositive, wrist=wnegative, fatherId=fReference[0]}
  [1186] = {x=31.104, y=0.000, z=-9.951, rx=-0.000, ry=0.000, rz=-0.000, shoulder=lefty, elbow=epositive, wrist=wnegative, fatherId=fReference[0]}
  [1187] = {x=31.641, y=0.000, z=-9.965, rx=-0.000, ry=0.000, rz=-0.000, shoulder=lefty, elbow=epositive, wrist=wnegative, fatherId=fReference[0]}
  [1188] = {x=31.502, y=0.000, z=-9.889, rx=-0.000, ry=0.000, rz=-0.000, shoulder=lefty, elbow=epositive, wrist=wnegative, fatherId=fReference[0]}
  [1189] = {x=30.889, y=0.000, z=-9.833, rx=-0.000, ry=0.000, rz=-0.000, shoulder=lefty, elbow=epositive, wrist=wnegative, fatherId=fReference[0]}
  [1190] = {x=30.349, y=0.000, z=-9.805, rx=-0.000, ry=0.000, rz=-0.000, shoulder=lefty, elbow=epositive, wrist=wnegative, fatherId=fReference[0]}
  [1191] = {x=29.821, y=0.000, z=-9.786, rx=-0.000, ry=0.000, rz=-0.000, shoulder=lefty, elbow=epositive, wrist=wnegative, fatherId=fReference[0]}
  [1192] = {x=29.301, y=0.000, z=-9.773, rx=-0.000, ry=0.000, rz=-0.000, shoulder=lefty, elbow=epositive, wrist=wnegative, fatherId=fReference[0]}
  [1193] = {x=28.786, y=0.000, z=-9.765, rx=-0.000, ry=0.000, rz=-0.000, shoulder=lefty, elbow=epositive, wrist=wnegative, fatherId=fReference[0]}
  [1194] = {x=28.274, y=0.000, z=-9.760, rx=-0.000, ry=0.000, rz=-0.000, shoulder=lefty, elbow=epositive, wrist=wnegative, fatherId=fReference[0]}
  [1195] = {x=27.763, y=0.000, z=-9.758, rx=-0.000, ry=0.000, rz=-0.000, shoulder=lefty, elbow=epositive, wrist=wnegative, fatherId=fReference[0]}
  [1196] = {x=27.255, y=0.000, z=-9.758, rx=-0.000, ry=0.000, rz=-0.000, shoulder=lefty, elbow=epositive, wrist=wnegative, fatherId=fReference[0]}
  [1197] = {x=26.748, y=0.000, z=-9.760, rx=-0.000, ry=0.000, rz=-0.000, shoulder=lefty, elbow=epositive, wrist=wnegative, fatherId=fReference[0]}
  [1198] = {x=26.242, y=0.000, z=-9.764, rx=-0.000, ry=0.000, rz=-0.000, shoulder=lefty, elbow=epositive, wrist=wnegative, fatherId=fReference[0]}
  [1199] = {x=25.737, y=0.000, z=-9.769, rx=-0.000, ry=0.000, rz=-0.000, shoulder=lefty, elbow=epositive, wrist=wnegative, fatherId=fReference[0]}
  [1200] = {x=25.232, y=0.000, z=-9.777, rx=-0.000, ry=0.000, rz=-0.000, shoulder=lefty, elbow=epositive, wrist=wnegative, fatherId=fReference[0]}
  [1201] = {x=24.728, y=0.000, z=-9.784, rx=-0.000, ry=0.000, rz=-0.000, shoulder=lefty, elbow=epositive, wrist=wnegative, fatherId=fReference[0]}
  [1202] = {x=24.224, y=0.000, z=-9.794, rx=-0.000, ry=0.000, rz=-0.000, shoulder=lefty, elbow=epositive, wrist=wnegative, fatherId=fReference[0]}
  [1203] = {x=23.723, y=0.000, z=-9.804, rx=-0.000, ry=0.000, rz=-0.000, shoulder=lefty, elbow=epositive, wrist=wnegative, fatherId=fReference[0]}
  [1204] = {x=23.223, y=0.000, z=-9.815, rx=-0.000, ry=0.000, rz=-0.000, shoulder=lefty, elbow=epositive, wrist=wnegative, fatherId=fReference[0]}
  [1205] = {x=22.721, y=0.000, z=-9.826, rx=-0.000, ry=0.000, rz=-0.000, shoulder=lefty, elbow=epositive, wrist=wnegative, fatherId=fReference[0]}
  [1206] = {x=22.220, y=0.000, z=-9.837, rx=-0.000, ry=0.000, rz=-0.000, shoulder=lefty, elbow=epositive, wrist=wnegative, fatherId=fReference[0]}
  [1207] = {x=21.720, y=0.000, z=-9.848, rx=-0.000, ry=0.000, rz=-0.000, shoulder=lefty, elbow=epositive, wrist=wnegative, fatherId=fReference[0]}
  [1208] = {x=21.220, y=0.000, z=-9.860, rx=-0.000, ry=0.000, rz=-0.000, shoulder=lefty, elbow=epositive, wrist=wnegative, fatherId=fReference[0]}
  [1209] = {x=20.719, y=0.000, z=-9.872, rx=-0.000, ry=0.000, rz=-0.000, shoulder=lefty, elbow=epositive, wrist=wnegative, fatherId=fReference[0]}
  [1210] = {x=20.219, y=0.000, z=-9.883, rx=-0.000, ry=0.000, rz=-0.000, shoulder=lefty, elbow=epositive, wrist=wnegative, fatherId=fReference[0]}
  [1211] = {x=19.718, y=0.000, z=-9.895, rx=-0.000, ry=0.000, rz=-0.000, shoulder=lefty, elbow=epositive, wrist=wnegative, fatherId=fReference[0]}
  [1212] = {x=19.217, y=0.000, z=-9.905, rx=-0.000, ry=0.000, rz=-0.000, shoulder=lefty, elbow=epositive, wrist=wnegative, fatherId=fReference[0]}
  [1213] = {x=18.717, y=0.000, z=-9.917, rx=-0.000, ry=0.000, rz=-0.000, shoulder=lefty, elbow=epositive, wrist=wnegative, fatherId=fReference[0]}
  [1214] = {x=18.216, y=0.000, z=-9.927, rx=-0.000, ry=0.000, rz=-0.000, shoulder=lefty, elbow=epositive, wrist=wnegative, fatherId=fReference[0]}
  [1215] = {x=17.715, y=0.000, z=-9.937, rx=-0.000, ry=0.000, rz=-0.000, shoulder=lefty, elbow=epositive, wrist=wnegative, fatherId=fReference[0]}
  [1216] = {x=17.214, y=0.000, z=-9.948, rx=-0.000, ry=0.000, rz=-0.000, shoulder=lefty, elbow=epositive, wrist=wnegative, fatherId=fReference[0]}
  [1217] = {x=16.714, y=0.000, z=-9.958, rx=-0.000, ry=0.000, rz=-0.000, shoulder=lefty, elbow=epositive, wrist=wnegative, fatherId=fReference[0]}
  [1218] = {x=16.212, y=0.000, z=-9.967, rx=-0.000, ry=0.000, rz=-0.000, shoulder=lefty, elbow=epositive, wrist=wnegative, fatherId=fReference[0]}
  [1219] = {x=15.711, y=0.000, z=-9.977, rx=-0.000, ry=0.000, rz=-0.000, shoulder=lefty, elbow=epositive, wrist=wnegative, fatherId=fReference[0]}
  [1220] = {x=15.210, y=0.000, z=-9.987, rx=-0.000, ry=0.000, rz=-0.000, shoulder=lefty, elbow=epositive, wrist=wnegative, fatherId=fReference[0]}
  [1221] = {x=14.709, y=0.000, z=-9.996, rx=-0.000, ry=0.000, rz=-0.000, shoulder=lefty, elbow=epositive, wrist=wnegative, fatherId=fReference[0]}
  [1222] = {x=14.207, y=0.000, z=-10.006, rx=-0.000, ry=0.000, rz=-0.000, shoulder=lefty, elbow=epositive, wrist=wnegative, fatherId=fReference[0]}
  [1223] = {x=13.706, y=0.000, z=-10.015, rx=-0.000, ry=0.000, rz=-0.000, shoulder=lefty, elbow=epositive, wrist=wnegative, fatherId=fReference[0]}
  [1224] = {x=13.204, y=0.000, z=-10.024, rx=-0.000, ry=0.000, rz=-0.000, shoulder=lefty, elbow=epositive, wrist=wnegative, fatherId=fReference[0]}
  [1225] = {x=12.702, y=0.000, z=-10.033, rx=-0.000, ry=0.000, rz=-0.000, shoulder=lefty, elbow=epositive, wrist=wnegative, fatherId=fReference[0]}
  [1226] = {x=12.200, y=0.000, z=-10.042, rx=-0.000, ry=0.000, rz=-0.000, shoulder=lefty, elbow=epositive, wrist=wnegative, fatherId=fReference[0]}
  [1227] = {x=11.698, y=0.000, z=-10.051, rx=-0.000, ry=0.000, rz=-0.000, shoulder=lefty, elbow=epositive, wrist=wnegative, fatherId=fReference[0]}
  [1228] = {x=11.196, y=0.000, z=-10.060, rx=-0.000, ry=0.000, rz=-0.000, shoulder=lefty, elbow=epositive, wrist=wnegative, fatherId=fReference[0]}
  [1229] = {x=10.694, y=0.000, z=-10.069, rx=-0.000, ry=0.000, rz=-0.000, shoulder=lefty, elbow=epositive, wrist=wnegative, fatherId=fReference[0]}
  [1230] = {x=10.191, y=0.000, z=-10.078, rx=-0.000, ry=0.000, rz=-0.000, shoulder=lefty, elbow=epositive, wrist=wnegative, fatherId=fReference[0]}
  [1231] = {x=9.688, y=0.000, z=-10.087, rx=-0.000, ry=0.000, rz=-0.000, shoulder=lefty, elbow=epositive, wrist=wnegative, fatherId=fReference[0]}
  [1232] = {x=9.186, y=0.000, z=-10.096, rx=-0.000, ry=0.000, rz=-0.000, shoulder=lefty, elbow=epositive, wrist=wnegative, fatherId=fReference[0]}
  [1233] = {x=8.684, y=0.000, z=-10.105, rx=-0.000, ry=0.000, rz=-0.000, shoulder=lefty, elbow=epositive, wrist=wnegative, fatherId=fReference[0]}
  [1234] = {x=8.182, y=0.000, z=-10.114, rx=-0.000, ry=0.000, rz=-0.000, shoulder=lefty, elbow=epositive, wrist=wnegative, fatherId=fReference[0]}
  [1235] = {x=7.680, y=0.000, z=-10.123, rx=-0.000, ry=0.000, rz=-0.000, shoulder=lefty, elbow=epositive, wrist=wnegative, fatherId=fReference[0]}
  [1236] = {x=7.177, y=0.000, z=-10.133, rx=-0.000, ry=0.000, rz=-0.000, shoulder=lefty, elbow=epositive, wrist=wnegative, fatherId=fReference[0]}
  [1237] = {x=6.674, y=0.000, z=-10.142, rx=-0.000, ry=0.000, rz=-0.000, shoulder=lefty, elbow=epositive, wrist=wnegative, fatherId=fReference[0]}
  [1238] = {x=6.172, y=0.000, z=-10.152, rx=-0.000, ry=0.000, rz=-0.000, shoulder=lefty, elbow=epositive, wrist=wnegative, fatherId=fReference[0]}
  [1239] = {x=5.669, y=0.000, z=-10.162, rx=-0.000, ry=0.000, rz=-0.000, shoulder=lefty, elbow=epositive, wrist=wnegative, fatherId=fReference[0]}
  [1240] = {x=5.166, y=0.000, z=-10.172, rx=-0.000, ry=0.000, rz=-0.000, shoulder=lefty, elbow=epositive, wrist=wnegative, fatherId=fReference[0]}
  [1241] = {x=4.663, y=0.000, z=-10.182, rx=-0.000, ry=0.000, rz=-0.000, shoulder=lefty, elbow=epositive, wrist=wnegative, fatherId=fReference[0]}
  [1242] = {x=4.161, y=0.000, z=-10.192, rx=-0.000, ry=0.000, rz=-0.000, shoulder=lefty, elbow=epositive, wrist=wnegative, fatherId=fReference[0]}
  [1243] = {x=3.658, y=0.000, z=-10.202, rx=-0.000, ry=0.000, rz=-0.000, shoulder=lefty, elbow=epositive, wrist=wnegative, fatherId=fReference[0]}
  [1244] = {x=3.155, y=0.000, z=-10.213, rx=-0.000, ry=0.000, rz=-0.000, shoulder=lefty, elbow=epositive, wrist=wnegative, fatherId=fReference[0]}
  [1245] = {x=2.651, y=0.000, z=-10.223, rx=-0.000, ry=0.000, rz=-0.000, shoulder=lefty, elbow=epositive, wrist=wnegative, fatherId=fReference[0]}
  [1246] = {x=2.147, y=0.000, z=-10.233, rx=-0.000, ry=0.000, rz=-0.000, shoulder=lefty, elbow=epositive, wrist=wnegative, fatherId=fReference[0]}
  [1247] = {x=1.644, y=0.000, z=-10.244, rx=-0.000, ry=0.000, rz=-0.000, shoulder=lefty, elbow=epositive, wrist=wnegative, fatherId=fReference[0]}
  [1248] = {x=1.141, y=0.000, z=-10.255, rx=-0.000, ry=0.000, rz=-0.000, shoulder=lefty, elbow=epositive, wrist=wnegative, fatherId=fReference[0]}
  [1249] = {x=0.638, y=0.000, z=-10.265, rx=-0.000, ry=0.000, rz=-0.000, shoulder=lefty, elbow=epositive, wrist=wnegative, fatherId=fReference[0]}
  [1250] = {x=0.136, y=0.000, z=-10.276, rx=-0.000, ry=0.000, rz=-0.000, shoulder=lefty, elbow=epositive, wrist=wnegative, fatherId=fReference[0]}
  [1251] = {x=-0.367, y=0.000, z=-10.286, rx=-0.000, ry=0.000, rz=-0.000, shoulder=lefty, elbow=epositive, wrist=wnegative, fatherId=fReference[0]}
  [1252] = {x=-0.869, y=0.000, z=-10.296, rx=-0.000, ry=0.000, rz=-0.000, shoulder=lefty, elbow=epositive, wrist=wnegative, fatherId=fReference[0]}
  [1253] = {x=-1.372, y=0.000, z=-10.306, rx=-0.000, ry=0.000, rz=-0.000, shoulder=lefty, elbow=epositive, wrist=wnegative, fatherId=fReference[0]}
  [1254] = {x=-1.875, y=0.000, z=-10.316, rx=-0.000, ry=0.000, rz=-0.000, shoulder=lefty, elbow=epositive, wrist=wnegative, fatherId=fReference[0]}
  [1255] = {x=-2.377, y=0.000, z=-10.326, rx=-0.000, ry=0.000, rz=-0.000, shoulder=lefty, elbow=epositive, wrist=wnegative, fatherId=fReference[0]}
  [1256] = {x=-2.879, y=0.000, z=-10.336, rx=-0.000, ry=0.000, rz=-0.000, shoulder=lefty, elbow=epositive, wrist=wnegative, fatherId=fReference[0]}
  [1257] = {x=-3.381, y=0.000, z=-10.346, rx=-0.000, ry=0.000, rz=-0.000, shoulder=lefty, elbow=epositive, wrist=wnegative, fatherId=fReference[0]}
  [1258] = {x=-3.883, y=0.000, z=-10.356, rx=-0.000, ry=0.000, rz=-0.000, shoulder=lefty, elbow=epositive, wrist=wnegative, fatherId=fReference[0]}
  [1259] = {x=-4.385, y=0.000, z=-10.366, rx=-0.000, ry=0.000, rz=-0.000, shoulder=lefty, elbow=epositive, wrist=wnegative, fatherId=fReference[0]}
  [1260] = {x=-4.888, y=0.000, z=-10.376, rx=-0.000, ry=0.000, rz=-0.000, shoulder=lefty, elbow=epositive, wrist=wnegative, fatherId=fReference[0]}
  [1261] = {x=-5.390, y=0.000, z=-10.386, rx=-0.000, ry=0.000, rz=-0.000, shoulder=lefty, elbow=epositive, wrist=wnegative, fatherId=fReference[0]}
  [1262] = {x=-5.893, y=0.000, z=-10.396, rx=-0.000, ry=0.000, rz=-0.000, shoulder=lefty, elbow=epositive, wrist=wnegative, fatherId=fReference[0]}
  [1263] = {x=-6.395, y=0.000, z=-10.405, rx=-0.000, ry=0.000, rz=-0.000, shoulder=lefty, elbow=epositive, wrist=wnegative, fatherId=fReference[0]}
  [1264] = {x=-6.897, y=0.000, z=-10.415, rx=-0.000, ry=0.000, rz=-0.000, shoulder=lefty, elbow=epositive, wrist=wnegative, fatherId=fReference[0]}
  [1265] = {x=-7.400, y=0.000, z=-10.424, rx=-0.000, ry=0.000, rz=-0.000, shoulder=lefty, elbow=epositive, wrist=wnegative, fatherId=fReference[0]}
  [1266] = {x=-7.902, y=0.000, z=-10.434, rx=-0.000, ry=0.000, rz=-0.000, shoulder=lefty, elbow=epositive, wrist=wnegative, fatherId=fReference[0]}
  [1267] = {x=-8.405, y=0.000, z=-10.443, rx=-0.000, ry=0.000, rz=-0.000, shoulder=lefty, elbow=epositive, wrist=wnegative, fatherId=fReference[0]}
  [1268] = {x=-8.907, y=0.000, z=-10.453, rx=-0.000, ry=0.000, rz=-0.000, shoulder=lefty, elbow=epositive, wrist=wnegative, fatherId=fReference[0]}
  [1269] = {x=-9.410, y=0.000, z=-10.464, rx=-0.000, ry=0.000, rz=-0.000, shoulder=lefty, elbow=epositive, wrist=wnegative, fatherId=fReference[0]}
  [1270] = {x=-9.913, y=0.000, z=-10.474, rx=-0.000, ry=0.000, rz=-0.000, shoulder=lefty, elbow=epositive, wrist=wnegative, fatherId=fReference[0]}
  [1271] = {x=-10.416, y=0.000, z=-10.484, rx=-0.000, ry=0.000, rz=-0.000, shoulder=lefty, elbow=epositive, wrist=wnegative, fatherId=fReference[0]}
  [1272] = {x=-10.919, y=0.000, z=-10.494, rx=-0.000, ry=0.000, rz=-0.000, shoulder=lefty, elbow=epositive, wrist=wnegative, fatherId=fReference[0]}
  [1273] = {x=-11.422, y=0.000, z=-10.504, rx=-0.000, ry=0.000, rz=-0.000, shoulder=lefty, elbow=epositive, wrist=wnegative, fatherId=fReference[0]}
  [1274] = {x=-11.926, y=0.000, z=-10.514, rx=-0.000, ry=0.000, rz=-0.000, shoulder=lefty, elbow=epositive, wrist=wnegative, fatherId=fReference[0]}
  [1275] = {x=-12.429, y=0.000, z=-10.524, rx=-0.000, ry=0.000, rz=-0.000, shoulder=lefty, elbow=epositive, wrist=wnegative, fatherId=fReference[0]}
  [1276] = {x=-12.932, y=0.000, z=-10.534, rx=-0.000, ry=0.000, rz=-0.000, shoulder=lefty, elbow=epositive, wrist=wnegative, fatherId=fReference[0]}
  [1277] = {x=-13.436, y=0.000, z=-10.545, rx=-0.000, ry=0.000, rz=-0.000, shoulder=lefty, elbow=epositive, wrist=wnegative, fatherId=fReference[0]}
  [1278] = {x=-13.939, y=0.000, z=-10.555, rx=-0.000, ry=0.000, rz=-0.000, shoulder=lefty, elbow=epositive, wrist=wnegative, fatherId=fReference[0]}
  [1279] = {x=-14.443, y=0.000, z=-10.566, rx=-0.000, ry=0.000, rz=-0.000, shoulder=lefty, elbow=epositive, wrist=wnegative, fatherId=fReference[0]}
  [1280] = {x=-14.947, y=0.000, z=-10.576, rx=-0.000, ry=0.000, rz=-0.000, shoulder=lefty, elbow=epositive, wrist=wnegative, fatherId=fReference[0]}
  [1281] = {x=-15.450, y=0.000, z=-10.587, rx=-0.000, ry=0.000, rz=-0.000, shoulder=lefty, elbow=epositive, wrist=wnegative, fatherId=fReference[0]}
  [1282] = {x=-15.954, y=0.000, z=-10.598, rx=-0.000, ry=0.000, rz=-0.000, shoulder=lefty, elbow=epositive, wrist=wnegative, fatherId=fReference[0]}
  [1283] = {x=-16.457, y=0.000, z=-10.609, rx=-0.000, ry=0.000, rz=-0.000, shoulder=lefty, elbow=epositive, wrist=wnegative, fatherId=fReference[0]}
  [1284] = {x=-16.959, y=0.000, z=-10.622, rx=-0.000, ry=0.000, rz=-0.000, shoulder=lefty, elbow=epositive, wrist=wnegative, fatherId=fReference[0]}
  [1285] = {x=-17.461, y=0.000, z=-10.635, rx=-0.000, ry=0.000, rz=-0.000, shoulder=lefty, elbow=epositive, wrist=wnegative, fatherId=fReference[0]}
  [1286] = {x=-17.967, y=0.000, z=-10.648, rx=-0.000, ry=0.000, rz=-0.000, shoulder=lefty, elbow=epositive, wrist=wnegative, fatherId=fReference[0]}
  [1287] = {x=-18.469, y=0.000, z=-10.661, rx=-0.000, ry=0.000, rz=-0.000, shoulder=lefty, elbow=epositive, wrist=wnegative, fatherId=fReference[0]}
  [1288] = {x=-18.968, y=0.000, z=-10.677, rx=-0.000, ry=0.000, rz=-0.000, shoulder=lefty, elbow=epositive, wrist=wnegative, fatherId=fReference[0]}
  [1289] = {x=-19.471, y=0.000, z=-10.693, rx=-0.000, ry=0.000, rz=-0.000, shoulder=lefty, elbow=epositive, wrist=wnegative, fatherId=fReference[0]}
  [1290] = {x=-19.971, y=0.000, z=-10.708, rx=-0.000, ry=0.000, rz=-0.000, shoulder=lefty, elbow=epositive, wrist=wnegative, fatherId=fReference[0]}
  [1291] = {x=-20.474, y=0.000, z=-10.723, rx=-0.000, ry=0.000, rz=-0.000, shoulder=lefty, elbow=epositive, wrist=wnegative, fatherId=fReference[0]}
  [1292] = {x=-20.978, y=0.000, z=-10.738, rx=-0.000, ry=0.000, rz=-0.000, shoulder=lefty, elbow=epositive, wrist=wnegative, fatherId=fReference[0]}
  [1293] = {x=-21.478, y=0.000, z=-10.756, rx=-0.000, ry=0.000, rz=-0.000, shoulder=lefty, elbow=epositive, wrist=wnegative, fatherId=fReference[0]}
  [1294] = {x=-21.984, y=0.000, z=-10.771, rx=-0.000, ry=0.000, rz=-0.000, shoulder=lefty, elbow=epositive, wrist=wnegative, fatherId=fReference[0]}
  [1295] = {x=-22.486, y=0.000, z=-10.788, rx=-0.000, ry=0.000, rz=-0.000, shoulder=lefty, elbow=epositive, wrist=wnegative, fatherId=fReference[0]}
  [1296] = {x=-22.987, y=0.000, z=-10.807, rx=-0.000, ry=0.000, rz=-0.000, shoulder=lefty, elbow=epositive, wrist=wnegative, fatherId=fReference[0]}
  [1297] = {x=-23.492, y=0.000, z=-10.825, rx=-0.000, ry=0.000, rz=-0.000, shoulder=lefty, elbow=epositive, wrist=wnegative, fatherId=fReference[0]}
  [1298] = {x=-23.998, y=0.000, z=-10.844, rx=-0.000, ry=0.000, rz=-0.000, shoulder=lefty, elbow=epositive, wrist=wnegative, fatherId=fReference[0]}
  [1299] = {x=-24.500, y=0.000, z=-10.865, rx=-0.000, ry=0.000, rz=-0.000, shoulder=lefty, elbow=epositive, wrist=wnegative, fatherId=fReference[0]}
  [1300] = {x=-25.008, y=0.000, z=-10.886, rx=-0.000, ry=0.000, rz=-0.000, shoulder=lefty, elbow=epositive, wrist=wnegative, fatherId=fReference[0]}
  [1301] = {x=-25.517, y=0.000, z=-10.907, rx=-0.000, ry=0.000, rz=-0.000, shoulder=lefty, elbow=epositive, wrist=wnegative, fatherId=fReference[0]}
  [1302] = {x=-26.027, y=0.000, z=-10.929, rx=-0.000, ry=0.000, rz=-0.000, shoulder=lefty, elbow=epositive, wrist=wnegative, fatherId=fReference[0]}
  [1303] = {x=-26.539, y=0.000, z=-10.954, rx=-0.000, ry=0.000, rz=-0.000, shoulder=lefty, elbow=epositive, wrist=wnegative, fatherId=fReference[0]}
  [1304] = {x=-27.056, y=0.000, z=-10.980, rx=-0.000, ry=0.000, rz=-0.000, shoulder=lefty, elbow=epositive, wrist=wnegative, fatherId=fReference[0]}
  [1305] = {x=-27.581, y=0.000, z=-11.009, rx=-0.000, ry=0.000, rz=-0.000, shoulder=lefty, elbow=epositive, wrist=wnegative, fatherId=fReference[0]}
  [1306] = {x=-28.109, y=0.000, z=-11.042, rx=-0.000, ry=0.000, rz=-0.000, shoulder=lefty, elbow=epositive, wrist=wnegative, fatherId=fReference[0]}
  [1307] = {x=-28.649, y=0.000, z=-11.075, rx=-0.000, ry=0.000, rz=-0.000, shoulder=lefty, elbow=epositive, wrist=wnegative, fatherId=fReference[0]}
  [1308] = {x=-29.185, y=0.000, z=-11.105, rx=-0.000, ry=0.000, rz=-0.000, shoulder=lefty, elbow=epositive, wrist=wnegative, fatherId=fReference[0]}
  [1309] = {x=-29.724, y=0.000, z=-11.126, rx=-0.000, ry=0.000, rz=-0.000, shoulder=lefty, elbow=epositive, wrist=wnegative, fatherId=fReference[0]}
  [1310] = {x=-30.224, y=0.000, z=-11.134, rx=-0.000, ry=0.000, rz=-0.000, shoulder=lefty, elbow=epositive, wrist=wnegative, fatherId=fReference[0]}
  [1311] = {x=-30.224, y=0.000, z=288.866, rx=-0.000, ry=0.000, rz=-0.000, shoulder=lefty, elbow=epositive, wrist=wnegative, fatherId=fReference[0]}
  [1312] = {x=-35.000, y=0.000, z=300.000, rx=-0.000, ry=0.000, rz=-0.000, shoulder=lefty, elbow=epositive, wrist=wnegative, fatherId=fReference[0]}
public tool tTool = {x=-0.414, y=-0.489, z=264.559, rx=180.000, ry=0.000, rz=-0.000, fatherId=flange[0], ioLink=valve1}
